(* CODESYS project tcunit.library
   Company: www.tcunit.org
   DefaultNamespace: TcUnit
   Version: 1.1.0.0
   Placeholder: TcUnit
   Author: Jakob Sagatowski and contributors
   Description: TwinCAT unit testing framework.
      Documentation and examples are available at www.tcunit.org
   Title: TcUnit

Project tree, tasks and I/O mapping:
  libraries: Base Interfaces, * (System); SysDir, * (System); SysFile, * (System); Tc2_Standard, * (Beckhoff Automation GmbH); Tc2_System, * (Beckhoff Automation GmbH); Tc2_Utilities, * (Beckhoff Automation GmbH)
  DUTs/
    data type E_AssertionType
    data type E_XmlError
    data type ST_AdsLogStringMessage
    data type ST_AssertArrayResult
    data type ST_AssertArrayResultInstances
    data type ST_AssertResult
    data type ST_AssertResultInstances
    data type ST_TestCaseResult
    data type ST_TestSuiteResult
    data type ST_TestSuiteResults
    data type U_ExpectedOrActual
  GVLs/
    global variables GVL_Param_TcUnit
    global variables GVL_TcUnit
  ITFs/
    interface I_AssertMessageFormatter: LogAssertFailure
    interface I_TestResultLogger: LogTestSuiteResults
    interface I_TestResults: GetAreTestResultsAvailable, GetTestSuiteResults
  POUs/
    Functions/
      WRITE_PROTECTED_/
        function WRITE_PROTECTED_BOOL [ST]
        function WRITE_PROTECTED_BYTE [ST]
        function WRITE_PROTECTED_DATE [ST]
        function WRITE_PROTECTED_DATE_AND_TIME [ST]
        function WRITE_PROTECTED_DINT [ST]
        function WRITE_PROTECTED_DWORD [ST]
        function WRITE_PROTECTED_INT [ST]
        function WRITE_PROTECTED_LINT [ST]
        function WRITE_PROTECTED_LREAL [ST]
        function WRITE_PROTECTED_LWORD [ST]
        function WRITE_PROTECTED_REAL [ST]
        function WRITE_PROTECTED_SINT [ST]
        function WRITE_PROTECTED_STRING [ST]
        function WRITE_PROTECTED_TIME [ST]
        function WRITE_PROTECTED_TIME_OF_DAY [ST]
        function WRITE_PROTECTED_UDINT [ST]
        function WRITE_PROTECTED_UINT [ST]
        function WRITE_PROTECTED_ULINT [ST]
        function WRITE_PROTECTED_USINT [ST]
        function WRITE_PROTECTED_WORD [ST]
        function WRITE_PROTECTED_WSTRING [ST]
      function F_AnyToUnionValue [ST]
      function F_AnyTypeClassToString [ST]
      function F_AssertionTypeToString [ST]
      function F_GetTestSuiteNameFromTestInstancePath [ST]
      function F_IsAnyEqualToUnionValue [ST]
      function F_RemoveInstancePathAndProjectNameFromTestInstancePath [ST]
      function IS_TEST_FINISHED [ST]
      function RUN [ST]
      function TEST [ST]
      function TEST_FINISHED [ST]
      function TEST_FINISHED_NAMED [ST]
    function block FB_AdjustAssertFailureMessageToMax253CharLength [ST]
    function block FB_AdsAssertMessageFormatter [ST]: LogAssertFailure
    function block FB_AdsLogStringMessageFifoQueue [ST]: GetAndRemoveLogFromQueue, GetLogCount, WriteLog
    function block FB_AdsTestResultLogger [ST]: FB_init, LogTestSuiteResults
    function block FB_AssertArrayResultStatic [ST]: AddAssertArrayResult, CopyDetectionCountAndResetDetectionCountInThisCycle, CreateAssertResultInstance, GetDetectionCount, GetDetectionCountThisCycle, GetNumberOfArrayAssertsForTest, ReportResult
    function block FB_AssertResultStatic [ST]: AddAssertResult, CopyDetectionCountAndResetDetectionCountInThisCycle, CreateAssertResultInstance, GetDetectionCount, GetDetectionCountThisCycle, GetNumberOfAssertsForTest, ReportResult
    function block FB_FileControl [ST]: Close, Delete, Open, Read, Write
    function block FB_StreamBuffer [ST]: Append, BufferSize, Clear, Copy, CutOff, Find, FindBack, Length, SetBuffer
    function block FB_TcUnitRunner [ST]: AbortRunningTestSuiteTests, RunTestSuiteTests
    function block FB_Test [ST]: GetAssertionMessage, GetAssertionType, GetName, GetNumberOfAssertions, IsFailed, IsFinished, IsSkipped, SetAssertionMessage, SetAssertionType, SetFailed, SetFinished, SetName, SetNumberOfAssertions, SetSkipped
    function block FB_TestResults [ST]: GetAreTestResultsAvailable, GetTestSuiteResults
    function block FB_TestSuite [ST]: AddTest, AddTestNameToInstancePath, AreAllTestsFinished, AssertArray2dEquals_LREAL, AssertArray2dEquals_REAL, AssertArray3dEquals_LREAL, AssertArray3dEquals_REAL, AssertArrayEquals_BOOL, AssertArrayEquals_BYTE, AssertArrayEquals_DINT, AssertArrayEquals_DWORD, AssertArrayEquals_INT, AssertArrayEquals_LINT, AssertArrayEquals_LREAL, AssertArrayEquals_LWORD, AssertArrayEquals_REAL, AssertArrayEquals_SINT, AssertArrayEquals_UDINT, AssertArrayEquals_UINT, AssertArrayEquals_ULINT, AssertArrayEquals_USINT, AssertArrayEquals_WORD, AssertEquals, AssertEquals_BOOL, AssertEquals_BYTE, AssertEquals_DATE, AssertEquals_DATE_AND_TIME, AssertEquals_DINT, AssertEquals_DWORD, AssertEquals_INT, AssertEquals_LINT, AssertEquals_LREAL, AssertEquals_LTIME, AssertEquals_LWORD, AssertEquals_REAL, AssertEquals_SINT, AssertEquals_STRING, AssertEquals_TIME, AssertEquals_TIME_OF_DAY, AssertEquals_UDINT, AssertEquals_UINT, AssertEquals_ULINT, AssertEquals_USINT, AssertEquals_WORD, AssertEquals_WSTRING, AssertFalse, AssertTrue, CalculateAndSetNumberOfAssertsForTest, FB_init, FindTestSuiteInstancePath, GetInstancePath, GetNumberOfFailedTests, GetNumberOfSkippedTests, GetNumberOfSuccessfulTests, GetNumberOfTests, GetTestByPosition, IsTestFinished, SetTestFailed, SetTestFinished
    function block FB_XmlControl [ST]: ClearBuffer, CloseTag, Length, NewComment, NewParameter, NewTag, NewTagData, SetBuffer, ToStartBuffer, WriteDocumentHeader
    function block FB_xUnitXmlPublisher [ST]: DeleteOpenWriteClose, FB_Init, Initialised, LogTestSuiteResults
  Version/
    global variables Global_Version
*)

// DUTs/E_AssertionType
{attribute 'qualified_only'}
{attribute 'strict'}
TYPE E_AssertionType :
(
    Type_UNDEFINED := 0,
    Type_ANY,

    (* Primitive types *)
    Type_BOOL,
    Type_BYTE,
    Type_DATE,
    Type_DATE_AND_TIME,
    Type_DINT,
    Type_DWORD,
    Type_INT,
    Type_LINT,
    Type_LREAL,
    Type_LTIME,
    Type_LWORD,
    Type_REAL,
    Type_SINT,
    Type_STRING,
    Type_TIME,
    Type_TIME_OF_DAY,
    Type_UDINT,
    Type_UINT,
    Type_ULINT,
    Type_USINT,
    Type_WORD,
    Type_WSTRING,

    (* Array types *)
    Type_Array2D_LREAL,
    Type_Array2D_REAL,
    Type_Array3D_LREAL,
    Type_Array3D_REAL,
    Type_Array_BOOL,
    Type_Array_BYTE,
    Type_Array_DINT,
    Type_Array_DWORD,
    Type_Array_INT,
    Type_Array_LINT,
    Type_Array_LREAL,
    Type_Array_LWORD,
    Type_Array_REAL,
    Type_Array_SINT,
    Type_Array_UDINT,
    Type_Array_UINT,
    Type_Array_ULINT,
    Type_Array_USINT,
    Type_Array_WORD
) BYTE;
END_TYPE

// DUTs/E_XmlError
{attribute 'qualified_only'}
{attribute 'strict'}
TYPE E_XmlError :
(
    Ok := 0,
    ErrorMaxBufferLen := 1,
    ErrorStringLen := 2,
    Error := 3
) BYTE;
END_TYPE

// DUTs/ST_AdsLogStringMessage
{attribute 'pack_mode' := '1'}
TYPE ST_AdsLogStringMessage :
STRUCT
	MsgCtrlMask : DWORD;
    MsgFmtStr : Tc2_System.T_MaxString;
    StrArg : Tc2_System.T_MaxString;
END_STRUCT
END_TYPE

// DUTs/ST_AssertArrayResult
TYPE ST_AssertArrayResult :
STRUCT
    ExpectedsSize : UDINT; // Size in bytes of the expecteds-array
    ExpectedsTypeClass : IBaseLibrary.TypeClass; // The data type of the expecteds-array
    ActualsSize : UDINT; // Size in bytes of the actuals-array
    ActualsTypeClass : IBaseLibrary.TypeClass; // The data type of the actuals-array
    Message : Tc2_System.T_MaxString;
    TestInstancePath : Tc2_System.T_MaxString;
END_STRUCT
END_TYPE

// DUTs/ST_AssertArrayResultInstances
TYPE ST_AssertArrayResultInstances :
STRUCT
    AssertArrayResult : ST_AssertArrayResult;
    DetectionCount : UINT; // Number of instances of the "AssertArrayResult"
    DetectionCountThisCycle : UINT; // Number of instance of the "AssertArrayResult" in this specific PLC-cycle
END_STRUCT
END_TYPE

// DUTs/ST_AssertResult
TYPE ST_AssertResult :
STRUCT
    Expected : U_ExpectedOrActual;
    Actual : U_ExpectedOrActual;
    Message : Tc2_System.T_MaxString;
    TestInstancePath : Tc2_System.T_MaxString;
END_STRUCT
END_TYPE

// DUTs/ST_AssertResultInstances
TYPE ST_AssertResultInstances :
STRUCT
    AssertResult : ST_AssertResult;
    DetectionCount : UINT; // Number of instances of the "AssertResult"
    DetectionCountThisCycle : UINT; // Number of instance of the "AssertResult" in this specific PLC-cycle
END_STRUCT
END_TYPE

// DUTs/ST_TestCaseResult
TYPE ST_TestCaseResult :
STRUCT
    TestName : Tc2_System.T_MaxString;
    TestClassName : Tc2_System.T_MaxString;
    TestIsFailed : BOOL;
    TestIsSkipped : BOOL;
    FailureMessage : Tc2_System.T_MaxString;
    FailureType : E_AssertionType;
    NumberOfAsserts : UINT;
END_STRUCT
END_TYPE

// DUTs/ST_TestSuiteResult
TYPE ST_TestSuiteResult :
STRUCT
    Name : Tc2_System.T_MaxString; // Full class name
    Identity : UINT(0..GVL_Param_TcUnit.MaxNumberOfTestSuites); // Should be 0..GVL_Param_TcUnit.MaxNumberOfTestSuites-1 but gives unknown compiler error
    NumberOfTests : UINT(0..GVL_Param_TcUnit.MaxNumberOfTestsForEachTestSuite);
    NumberOfFailedTests : UINT(0..GVL_Param_TcUnit.MaxNumberOfTestsForEachTestSuite);
    TestCaseResults : ARRAY[1..GVL_Param_TcUnit.MaxNumberOfTestsForEachTestSuite] OF ST_TestCaseResult;
END_STRUCT
END_TYPE

// DUTs/ST_TestSuiteResults
TYPE ST_TestSuiteResults :
STRUCT
    (* General test results *)
    NumberOfTestSuites : UINT; // The total number of test suites
    NumberOfTestCases : UINT; // The total number of test cases (for all test suites)
    NumberOfSuccessfulTestCases : UINT; // The total number of test cases that had all ASSERTS successful
    NumberOfFailedTestCases : UINT; // The total number of test cases that had at least one ASSERT failed

    (* Test results for each individiual test suite *)
    TestSuiteResults : ARRAY[1..GVL_Param_TcUnit.MaxNumberOfTestSuites] OF ST_TestSuiteResult;
END_STRUCT
END_TYPE

// DUTs/U_ExpectedOrActual
TYPE U_ExpectedOrActual :
UNION
    boolExpectedOrActual : BOOL;
    bitExpectedOrActual : BIT;
    byteExpectedOrActual : BYTE;
    dwordExpectedOrActual : DWORD;
    lwordExpectedOrActual : LWORD;
    stringExpectedOrActual : Tc2_System.T_MaxString;
    udintExpectedOrActual : UDINT;
    uintExpectedOrActual : UINT;
    usintExpectedOrActual : USINT;
    sintExpectedOrActual : SINT;
    intExpectedOrActual : INT;
    wordExpectedOrActual : WORD;
    dintExpectedOrActual : DINT;
    lintExpectedOrActual : LINT;
    ulintExpectedOrActual : ULINT;
    realExpectedOrActual : REAL;
    lrealExpectedOrActual : LREAL;
    wstringExpectedOrActual : WSTRING(255);
    timeExpectedOrActual : TIME;
    ltimeExpectedOrActual : LTIME;
    dateExpectedOrActual : DATE;
    dateandtimeExpectedOrActual : DATE_AND_TIME;
    timeofdayExpectedOrActual : TIME_OF_DAY;
END_UNION
END_TYPE

// GVLs/GVL_Param_TcUnit
{attribute 'qualified_only'}
VAR_GLOBAL CONSTANT
    MaxNumberOfTestSuites : UINT := 1000;
    MaxNumberOfTestsForEachTestSuite : UINT := 100;
    MaxNumberOfAssertsForEachTestSuite : UINT := 1000;

    (* TcUnit logs complete test results. These include:
         - Number of test suites
         - Number of tests
         - Number of successful tests
         - Number of failed tests
         - Any eventual failed assertion (with the expected & actual value plus an user defined message)
       These are all printed to the ADS logger (Visual Studio error list) marked with ERROR criticality

       On top of this TcUnit also reports some statistics/extended information with HINT/INFO criticality.
       These statistics are more detailed results of the tests. This information is used when results are
       being collected by an external software (such as TcUnit-Runner) to do for example Jenkins integration.
       This extra information however takes time to print, so by setting the following parameter to FALSE
       it will speed up TcUnit finishing. *)
    LogExtendedResults : BOOL := TRUE;

    (* Enable (TRUE) or disable (FALSE) publishing of the xUnit Xml report *)
    xUnitEnablePublish : BOOL := FALSE;

    (* Default reserved PLC memory buffer used for composition of the xUnit xml file (64 kb default) *)
    xUnitBufferSize : UDINT := 65535;

    (* Default path and filename for the xunit testresults e.g.: for use with jenkins *)
    xUnitFilePath : Tc2_System.T_MaxString := 'C:\tcunit_xunit_testresults.xml';

    (* This is the maximum number of ADS-messages that can be stored for reporting at the same time.
       Having a size of 2000 means that it's possible to report up to ~400 test cases in one single
       PLC cycle. Each entry consumes around 500 bytes, so with an example of a ring buffer size of
       2000 it means that TcUnit will consume around 1 MB of router memory. *) 
    AdsLogMessageFifoRingBufferSize : UINT := 2000;
END_VAR

// GVLs/GVL_TcUnit
{attribute 'no_assign'}
{attribute 'qualified_only'}
VAR_GLOBAL
    TcUnitRunner : FB_TcUnitRunner;

    (* Indication of whether the last instantiated test suite has an assert instance created *)
    TestSuiteIsRegistered : BOOL;

    (* Pointer to current test suite being called *)
    CurrentTestSuiteBeingCalled : POINTER TO FB_TestSuite;

    (* Current name of test being called *)
    CurrentTestNameBeingCalled : Tc2_System.T_MaxString;

    (* Whether or not the current test being called has finished running *)
    CurrentTestIsFinished : BOOL;

    (* This is a flag that indicates that the current test should be ignored, and
       thus that all assertions under it should be ignored as well. A test can be ignored either
       because the user has requested so, or because the test is a duplicate name *)
    IgnoreCurrentTest : BOOL;

    (* The assert function block instance should be 1:1 mapped to
       the test suite instance path. *)
    NumberOfInitializedTestSuites : UINT := 0;
    TestSuiteAddresses : ARRAY[1..GVL_Param_TcUnit.MaxNumberOfTestSuites] OF POINTER TO FB_TestSuite;

    (* Buffered ADS message queue for output to the error list *)
    AdsMessageQueue : FB_AdsLogStringMessageFifoQueue;
END_VAR

// Version/Global_Version
{attribute 'TcGenerated'}
{attribute 'no-analysis'}
{attribute 'linkalways'}
// This function has been automatically generated from the project information.
VAR_GLOBAL CONSTANT
	{attribute 'const_non_replaced'}
	stLibVersion_TcUnit : ST_LibVersion := (iMajor := 1, iMinor := 1, iBuild := 0, iRevision := 0, sVersion := '1.1.0.0');
END_VAR

// ITFs/I_AssertMessageFormatter
INTERFACE I_AssertMessageFormatter

METHOD LogAssertFailure
VAR_INPUT
    Expected : Tc2_System.T_MaxString;
    Actual : Tc2_System.T_MaxString;
    Message : Tc2_System.T_MaxString;
    TestInstancePath : Tc2_System.T_MaxString;
END_VAR
END_METHOD

END_INTERFACE

// ITFs/I_TestResultLogger
INTERFACE I_TestResultLogger

METHOD PUBLIC LogTestSuiteResults
END_METHOD

END_INTERFACE

// ITFs/I_TestResults
INTERFACE I_TestResults

METHOD GetAreTestResultsAvailable : BOOL
END_METHOD

METHOD GetTestSuiteResults : REFERENCE TO ST_TestSuiteResults;
END_METHOD

END_INTERFACE

// POUs/Functions/WRITE_PROTECTED_/WRITE_PROTECTED_BOOL
FUNCTION WRITE_PROTECTED_BOOL
VAR_INPUT
    Ptr : POINTER TO BOOL;
    Value : BOOL;
END_VAR

Ptr^ := Value;

END_FUNCTION

// POUs/Functions/WRITE_PROTECTED_/WRITE_PROTECTED_BYTE
FUNCTION WRITE_PROTECTED_BYTE
VAR_INPUT
    Ptr : POINTER TO BYTE;
    Value : BYTE;
END_VAR

Ptr^ := Value;

END_FUNCTION

// POUs/Functions/WRITE_PROTECTED_/WRITE_PROTECTED_DATE
FUNCTION WRITE_PROTECTED_DATE
VAR_INPUT
    Ptr : POINTER TO DATE;
    Value : DATE;
END_VAR

Ptr^ := Value;

END_FUNCTION

// POUs/Functions/WRITE_PROTECTED_/WRITE_PROTECTED_DATE_AND_TIME
FUNCTION WRITE_PROTECTED_DATE_AND_TIME
VAR_INPUT
    Ptr : POINTER TO DATE_AND_TIME;
    Value : DATE_AND_TIME;
END_VAR

Ptr^ := Value;

END_FUNCTION

// POUs/Functions/WRITE_PROTECTED_/WRITE_PROTECTED_DINT
FUNCTION WRITE_PROTECTED_DINT
VAR_INPUT
    Ptr : POINTER TO DINT;
    Value : DINT;
END_VAR

Ptr^ := Value;

END_FUNCTION

// POUs/Functions/WRITE_PROTECTED_/WRITE_PROTECTED_DWORD
FUNCTION WRITE_PROTECTED_DWORD
VAR_INPUT
    Ptr : POINTER TO DWORD;
    Value : DWORD;
END_VAR

Ptr^ := Value;

END_FUNCTION

// POUs/Functions/WRITE_PROTECTED_/WRITE_PROTECTED_INT
FUNCTION WRITE_PROTECTED_INT
VAR_INPUT
    Ptr : POINTER TO INT;
    Value : INT;
END_VAR

Ptr^ := Value;

END_FUNCTION

// POUs/Functions/WRITE_PROTECTED_/WRITE_PROTECTED_LINT
FUNCTION WRITE_PROTECTED_LINT
VAR_INPUT
    Ptr : POINTER TO LINT;
    Value : LINT;
END_VAR

Ptr^ := Value;

END_FUNCTION

// POUs/Functions/WRITE_PROTECTED_/WRITE_PROTECTED_LREAL
FUNCTION WRITE_PROTECTED_LREAL
VAR_INPUT
    Ptr : POINTER TO LREAL;
    Value : LREAL;
END_VAR

Ptr^ := Value;

END_FUNCTION

// POUs/Functions/WRITE_PROTECTED_/WRITE_PROTECTED_LWORD
FUNCTION WRITE_PROTECTED_LWORD
VAR_INPUT
    Ptr : POINTER TO LWORD;
    Value : LWORD;
END_VAR

Ptr^ := Value;

END_FUNCTION

// POUs/Functions/WRITE_PROTECTED_/WRITE_PROTECTED_REAL
FUNCTION WRITE_PROTECTED_REAL
VAR_INPUT
    Ptr : POINTER TO REAL;
    Value : REAL;
END_VAR

Ptr^ := Value;

END_FUNCTION

// POUs/Functions/WRITE_PROTECTED_/WRITE_PROTECTED_SINT
FUNCTION WRITE_PROTECTED_SINT
VAR_INPUT
    Ptr : POINTER TO SINT;
    Value : SINT;
END_VAR

Ptr^ := Value;

END_FUNCTION

// POUs/Functions/WRITE_PROTECTED_/WRITE_PROTECTED_STRING
FUNCTION WRITE_PROTECTED_STRING
VAR_INPUT
    Ptr : POINTER TO STRING;
    Value : STRING;
END_VAR

Ptr^ := Value;

END_FUNCTION

// POUs/Functions/WRITE_PROTECTED_/WRITE_PROTECTED_TIME
FUNCTION WRITE_PROTECTED_TIME
VAR_INPUT
    Ptr : POINTER TO TIME;
    Value : TIME;
END_VAR

Ptr^ := Value;

END_FUNCTION

// POUs/Functions/WRITE_PROTECTED_/WRITE_PROTECTED_TIME_OF_DAY
FUNCTION WRITE_PROTECTED_TIME_OF_DAY
VAR_INPUT
    Ptr : POINTER TO TIME_OF_DAY;
    Value : TIME_OF_DAY;
END_VAR

Ptr^ := Value;

END_FUNCTION

// POUs/Functions/WRITE_PROTECTED_/WRITE_PROTECTED_UDINT
FUNCTION WRITE_PROTECTED_UDINT
VAR_INPUT
    Ptr : POINTER TO UDINT;
    Value : UDINT;
END_VAR

Ptr^ := Value;

END_FUNCTION

// POUs/Functions/WRITE_PROTECTED_/WRITE_PROTECTED_UINT
FUNCTION WRITE_PROTECTED_UINT
VAR_INPUT
    Ptr : POINTER TO UINT;
    Value : UINT;
END_VAR

Ptr^ := Value;

END_FUNCTION

// POUs/Functions/WRITE_PROTECTED_/WRITE_PROTECTED_ULINT
FUNCTION WRITE_PROTECTED_ULINT
VAR_INPUT
    Ptr : POINTER TO ULINT;
    Value : ULINT;
END_VAR

Ptr^ := Value;

END_FUNCTION

// POUs/Functions/WRITE_PROTECTED_/WRITE_PROTECTED_USINT
FUNCTION WRITE_PROTECTED_USINT
VAR_INPUT
    Ptr : POINTER TO USINT;
    Value : USINT;
END_VAR

Ptr^ := Value;

END_FUNCTION

// POUs/Functions/WRITE_PROTECTED_/WRITE_PROTECTED_WORD
FUNCTION WRITE_PROTECTED_WORD
VAR_INPUT
    Ptr : POINTER TO WORD;
    Value : WORD;
END_VAR

Ptr^ := Value;

END_FUNCTION

// POUs/Functions/WRITE_PROTECTED_/WRITE_PROTECTED_WSTRING
FUNCTION WRITE_PROTECTED_WSTRING
VAR_INPUT
    Ptr : POINTER TO WSTRING;
    Value : WSTRING;
END_VAR

Ptr^ := Value;

END_FUNCTION

// POUs/Functions/F_AnyToUnionValue
FUNCTION F_AnyToUnionValue : U_ExpectedOrActual
VAR_INPUT
    AnySize : UDINT;
    AnyTypeClass : IBaseLibrary.TypeClass;
    AnyValue : POINTER TO BYTE;
END_VAR

CASE AnyTypeClass OF
    IBaseLibrary.TypeClass.TYPE_BOOL :
        Tc2_System.MEMCPY(destaddr := ADR(F_AnyToUnionValue.boolExpectedOrActual),
                          srcAddr := AnyValue,
                          n := AnySize);

    IBaseLibrary.TypeClass.TYPE_BIT :
        {warning disable C0355}
        Tc2_System.MEMCPY(destaddr := ADR(F_AnyToUnionValue.bitExpectedOrActual),
                          srcAddr := AnyValue,
                          n := AnySize);
        {warning enable C0355}

    IBaseLibrary.TypeClass.TYPE_BYTE :
        Tc2_System.MEMCPY(destaddr := ADR(F_AnyToUnionValue.byteExpectedOrActual),
                          srcAddr := AnyValue,
                          n := AnySize);

    IBaseLibrary.TypeClass.TYPE_WORD :
        Tc2_System.MEMCPY(destaddr := ADR(F_AnyToUnionValue.wordExpectedOrActual),
                          srcAddr := AnyValue,
                          n := AnySize);

    IBaseLibrary.TypeClass.TYPE_DWORD :
        Tc2_System.MEMCPY(destaddr := ADR(F_AnyToUnionValue.dwordExpectedOrActual),
                          srcAddr := AnyValue,
                          n := AnySize);

    IBaseLibrary.TypeClass.TYPE_LWORD :
        Tc2_System.MEMCPY(destaddr := ADR(F_AnyToUnionValue.lwordExpectedOrActual),
                          srcAddr := AnyValue,
                          n := AnySize);

    IBaseLibrary.TypeClass.TYPE_SINT :
        Tc2_System.MEMCPY(destaddr := ADR(F_AnyToUnionValue.sintExpectedOrActual),
                          srcAddr := AnyValue,
                          n := AnySize);

    IBaseLibrary.TypeClass.TYPE_INT :
        Tc2_System.MEMCPY(destaddr := ADR(F_AnyToUnionValue.intExpectedOrActual),
                          srcAddr := AnyValue,
                          n := AnySize);

    IBaseLibrary.TypeClass.TYPE_DINT :
        Tc2_System.MEMCPY(destaddr := ADR(F_AnyToUnionValue.dintExpectedOrActual),
                          srcAddr := AnyValue,
                          n := AnySize);

    IBaseLibrary.TypeClass.TYPE_LINT :
        Tc2_System.MEMCPY(destaddr := ADR(F_AnyToUnionValue.lintExpectedOrActual),
                          srcAddr := AnyValue,
                          n := AnySize);

    IBaseLibrary.TypeClass.TYPE_USINT :
        Tc2_System.MEMCPY(destaddr := ADR(F_AnyToUnionValue.usintExpectedOrActual),
                          srcAddr := AnyValue,
                          n := AnySize);

    IBaseLibrary.TypeClass.TYPE_UINT :
        Tc2_System.MEMCPY(destaddr := ADR(F_AnyToUnionValue.uintExpectedOrActual),
                          srcAddr := AnyValue,
                          n := AnySize);

    IBaseLibrary.TypeClass.TYPE_UDINT :
        Tc2_System.MEMCPY(destaddr := ADR(F_AnyToUnionValue.udintExpectedOrActual),
                          srcAddr := AnyValue,
                          n := AnySize);

    IBaseLibrary.TypeClass.TYPE_ULINT :
        Tc2_System.MEMCPY(destaddr := ADR(F_AnyToUnionValue.ulintExpectedOrActual),
                          srcAddr := AnyValue,
                          n := AnySize);

    IBaseLibrary.TypeClass.TYPE_REAL :
        Tc2_System.MEMCPY(destaddr := ADR(F_AnyToUnionValue.realExpectedOrActual),
                          srcAddr := AnyValue,
                          n := AnySize);

    IBaseLibrary.TypeClass.TYPE_LREAL :
        Tc2_System.MEMCPY(destaddr := ADR(F_AnyToUnionValue.lrealExpectedOrActual),
                          srcAddr := AnyValue,
                          n := AnySize);

    IBaseLibrary.TypeClass.TYPE_STRING :
        Tc2_System.MEMCPY(destaddr := ADR(F_AnyToUnionValue.stringExpectedOrActual),
                          srcAddr := AnyValue,
                          n := AnySize);

    IBaseLibrary.TypeClass.TYPE_WSTRING :
        Tc2_System.MEMCPY(destaddr := ADR(F_AnyToUnionValue.wstringExpectedOrActual),
                          srcAddr := AnyValue,
                          n := AnySize);

    IBaseLibrary.TypeClass.TYPE_TIME :
        Tc2_System.MEMCPY(destaddr := ADR(F_AnyToUnionValue.timeExpectedOrActual),
                          srcAddr := AnyValue,
                          n := AnySize);

    IBaseLibrary.TypeClass.TYPE_DATE :
        Tc2_System.MEMCPY(destaddr := ADR(F_AnyToUnionValue.dateExpectedOrActual),
                          srcAddr := AnyValue,
                          n := AnySize);

    IBaseLibrary.TypeClass.TYPE_DATEANDTIME :
        Tc2_System.MEMCPY(destaddr := ADR(F_AnyToUnionValue.dateandtimeExpectedOrActual),
                          srcAddr := AnyValue,
                          n := AnySize);

    IBaseLibrary.TypeClass.TYPE_TIMEOFDAY :
        Tc2_System.MEMCPY(destaddr := ADR(F_AnyToUnionValue.timeofdayExpectedOrActual),
                          srcAddr := AnyValue,
                          n := AnySize);

    IBaseLibrary.TypeClass.TYPE_POINTER :
        (* None *)

    IBaseLibrary.TypeClass.TYPE_REFERENCE :
        (* None *)

    IBaseLibrary.TypeClass.TYPE_SUBRANGE :
        (* None *)

    IBaseLibrary.TypeClass.TYPE_ENUM :
        (* None *)

    IBaseLibrary.TypeClass.TYPE_ARRAY :
        (* None *)

    IBaseLibrary.TypeClass.TYPE_PARAMS :
        (* None *)

    IBaseLibrary.TypeClass.TYPE_USERDEF :
        (* None *)

    IBaseLibrary.TypeClass.TYPE_NONE :
        (* None *)

    IBaseLibrary.TypeClass.TYPE_ANY :
        (* None *)

    IBaseLibrary.TypeClass.TYPE_ANYBIT :
        (* None *)

    IBaseLibrary.TypeClass.TYPE_ANYDATE :
        (* None *)

    IBaseLibrary.TypeClass.TYPE_ANYINT :
        (* None *)

    IBaseLibrary.TypeClass.TYPE_ANYNUM :
        (* None *)

    IBaseLibrary.TypeClass.TYPE_ANYREAL :
        (* None *)

    IBaseLibrary.TypeClass.TYPE_LAZY :
        (* None *)

    IBaseLibrary.TypeClass.TYPE_LTIME :
        Tc2_System.MEMCPY(destaddr := ADR(F_AnyToUnionValue.ltimeExpectedOrActual),
                          srcAddr := AnyValue,
                          n := AnySize);

    IBaseLibrary.TypeClass.TYPE_BITCONST :
        (* None *)

    IBaseLibrary.TypeClass.TYPE_INTERFACE :
        (* None *)

    ELSE
        (* None *)
END_CASE

END_FUNCTION

// POUs/Functions/F_AnyTypeClassToString
(*
    This function takes the type-class of a ANY-variable and returns the STRING representation of it.
*)
FUNCTION F_AnyTypeClassToString : STRING
VAR_INPUT
    AnyTypeClass : __SYSTEM.TYPE_CLASS;
END_VAR

CASE UDINT_TO_INT(AnyTypeClass) OF
    IBaseLibrary.TypeClass.TYPE_BOOL :
        F_AnyTypeClassToString := 'BOOL';
    IBaseLibrary.TypeClass.TYPE_BIT :
        F_AnyTypeClassToString := 'BIT';
    IBaseLibrary.TypeClass.TYPE_BYTE :
        F_AnyTypeClassToString := 'BYTE';
    IBaseLibrary.TypeClass.TYPE_WORD :
        F_AnyTypeClassToString := 'WORD';
    IBaseLibrary.TypeClass.TYPE_DWORD :
        F_AnyTypeClassToString := 'DWORD';
    IBaseLibrary.TypeClass.TYPE_LWORD :
        F_AnyTypeClassToString := 'LWORD';
    IBaseLibrary.TypeClass.TYPE_SINT :
        F_AnyTypeClassToString := 'SINT';
    IBaseLibrary.TypeClass.TYPE_INT :
        F_AnyTypeClassToString := 'INT';
    IBaseLibrary.TypeClass.TYPE_DINT :
        F_AnyTypeClassToString := 'DINT';
    IBaseLibrary.TypeClass.TYPE_LINT :
        F_AnyTypeClassToString := 'LINT';
    IBaseLibrary.TypeClass.TYPE_USINT :
        F_AnyTypeClassToString := 'USINT';
    IBaseLibrary.TypeClass.TYPE_UINT :
        F_AnyTypeClassToString := 'UINT';
    IBaseLibrary.TypeClass.TYPE_UDINT :
        F_AnyTypeClassToString := 'UDINT';
    IBaseLibrary.TypeClass.TYPE_ULINT :
        F_AnyTypeClassToString := 'ULINT';
    IBaseLibrary.TypeClass.TYPE_REAL :
        F_AnyTypeClassToString := 'REAL';
    IBaseLibrary.TypeClass.TYPE_LREAL :
        F_AnyTypeClassToString := 'LREAL';
    IBaseLibrary.TypeClass.TYPE_STRING :
        F_AnyTypeClassToString := 'STRING';
    IBaseLibrary.TypeClass.TYPE_WSTRING :
        F_AnyTypeClassToString := 'WSTRING';
    IBaseLibrary.TypeClass.TYPE_TIME :
        F_AnyTypeClassToString := 'TIME';
    IBaseLibrary.TypeClass.TYPE_DATE :
        F_AnyTypeClassToString := 'DATE';
    IBaseLibrary.TypeClass.TYPE_DATEANDTIME :
        F_AnyTypeClassToString := 'DATEANDTIME';
    IBaseLibrary.TypeClass.TYPE_TIMEOFDAY :
        F_AnyTypeClassToString := 'TIMEOFDAY';
    IBaseLibrary.TypeClass.TYPE_POINTER :
        F_AnyTypeClassToString := 'POINTER';
    IBaseLibrary.TypeClass.TYPE_REFERENCE :
        F_AnyTypeClassToString := 'REFERENCE';
    IBaseLibrary.TypeClass.TYPE_SUBRANGE :
        F_AnyTypeClassToString := 'SUBRANGE';
    IBaseLibrary.TypeClass.TYPE_ENUM :
        F_AnyTypeClassToString := 'ENUM';
    IBaseLibrary.TypeClass.TYPE_ARRAY :
        F_AnyTypeClassToString := 'ARRAY';
    IBaseLibrary.TypeClass.TYPE_PARAMS :
        F_AnyTypeClassToString := 'PARAMS';
    IBaseLibrary.TypeClass.TYPE_USERDEF :
        F_AnyTypeClassToString := 'USERDEF';
    IBaseLibrary.TypeClass.TYPE_NONE :
        F_AnyTypeClassToString := 'NONE';
    IBaseLibrary.TypeClass.TYPE_ANY :
        F_AnyTypeClassToString := 'ANY';
    IBaseLibrary.TypeClass.TYPE_ANYBIT :
        F_AnyTypeClassToString := 'ANYBIT';
    IBaseLibrary.TypeClass.TYPE_ANYDATE :
        F_AnyTypeClassToString := 'ANYDATE';
    IBaseLibrary.TypeClass.TYPE_ANYINT :
        F_AnyTypeClassToString := 'ANYINT';
    IBaseLibrary.TypeClass.TYPE_ANYNUM :
        F_AnyTypeClassToString := 'ANYNUM';
    IBaseLibrary.TypeClass.TYPE_ANYREAL :
        F_AnyTypeClassToString := 'ANYREAL';
    IBaseLibrary.TypeClass.TYPE_LAZY :
        F_AnyTypeClassToString := 'LAZY';
    IBaseLibrary.TypeClass.TYPE_LTIME :
        F_AnyTypeClassToString := 'LTIME';
    IBaseLibrary.TypeClass.TYPE_BITCONST :
        F_AnyTypeClassToString := 'BITCONST';
    IBaseLibrary.TypeClass.TYPE_INTERFACE :
        F_AnyTypeClassToString := 'INTERFACE';
    ELSE
        F_AnyTypeClassToString := 'UNKNOWN';
END_CASE

END_FUNCTION

// POUs/Functions/F_AssertionTypeToString
(* Since TwinCAT 3.1.4024.x it's possible to do TO_STRING on enumerations,
   but for backward compability we need to do it manually *)
FUNCTION F_AssertionTypeToString : Tc2_System.T_MaxString
VAR_INPUT
    AssertionType : E_AssertionType;
END_VAR

CASE AssertionType OF
    E_AssertionType.Type_UNDEFINED :
        F_AssertionTypeToString := 'UNDEFINED';
    E_AssertionType.Type_ANY :
        F_AssertionTypeToString := 'ANY';

    (* Primitive types *)
    E_AssertionType.Type_BOOL :
        F_AssertionTypeToString := 'BOOL';
    E_AssertionType.Type_BYTE :
        F_AssertionTypeToString := 'BYTE';
    E_AssertionType.Type_DATE :
        F_AssertionTypeToString := 'DATE';
    E_AssertionType.Type_DATE_AND_TIME :
        F_AssertionTypeToString := 'DATE_AND_TIME';
    E_AssertionType.Type_DINT :
        F_AssertionTypeToString := 'DINT';
    E_AssertionType.Type_DWORD :
        F_AssertionTypeToString := 'DWORD';
    E_AssertionType.Type_INT :
        F_AssertionTypeToString := 'INT';
    E_AssertionType.Type_LINT :
        F_AssertionTypeToString := 'LINT';
    E_AssertionType.Type_LREAL :
        F_AssertionTypeToString := 'LREAL';
    E_AssertionType.Type_LTIME :
        F_AssertionTypeToString := 'LTIME';
    E_AssertionType.Type_LWORD :
        F_AssertionTypeToString := 'LWORD';
    E_AssertionType.Type_REAL :
        F_AssertionTypeToString := 'REAL';
    E_AssertionType.Type_SINT :
        F_AssertionTypeToString := 'SINT';
    E_AssertionType.Type_STRING :
        F_AssertionTypeToString := 'STRING';
    E_AssertionType.Type_TIME :
        F_AssertionTypeToString := 'TIME';
    E_AssertionType.Type_TIME_OF_DAY :
        F_AssertionTypeToString := 'TIME_OF_DAY';
    E_AssertionType.Type_UDINT :
        F_AssertionTypeToString := 'UDINT';
    E_AssertionType.Type_UINT :
        F_AssertionTypeToString := 'UINT';
    E_AssertionType.Type_ULINT :
        F_AssertionTypeToString := 'ULINT';
    E_AssertionType.Type_USINT :
        F_AssertionTypeToString := 'USINT';
    E_AssertionType.Type_WORD :
        F_AssertionTypeToString := 'WORD';
    E_AssertionType.Type_WSTRING :
        F_AssertionTypeToString := 'WSTRING';


    (* Array types *)
    E_AssertionType.Type_Array2D_LREAL :
        F_AssertionTypeToString := 'Array2D_LREAL';
    E_AssertionType.Type_Array2D_REAL :
        F_AssertionTypeToString := 'Array2D_REAL';
    E_AssertionType.Type_Array3D_LREAL :
        F_AssertionTypeToString := 'Array3D_LREAL';
    E_AssertionType.Type_Array3D_REAL :
        F_AssertionTypeToString := 'Array3D_REAL';
    E_AssertionType.Type_Array_BOOL :
        F_AssertionTypeToString := 'Array_BOOL';
    E_AssertionType.Type_Array_BYTE :
        F_AssertionTypeToString := 'Array_BYTE';
    E_AssertionType.Type_Array_DINT :
        F_AssertionTypeToString := 'Array_DINT';
    E_AssertionType.Type_Array_DWORD :
        F_AssertionTypeToString := 'Array_DWORD';
    E_AssertionType.Type_Array_INT :
        F_AssertionTypeToString := 'Array_INT';
    E_AssertionType.Type_Array_LINT :
        F_AssertionTypeToString := 'Array_LINT';
    E_AssertionType.Type_Array_LREAL :
        F_AssertionTypeToString := 'Array_LREAL';
    E_AssertionType.Type_Array_LWORD :
        F_AssertionTypeToString := 'Array_LWORD';
    E_AssertionType.Type_Array_REAL :
        F_AssertionTypeToString := 'Array_REAL';
    E_AssertionType.Type_Array_SINT :
        F_AssertionTypeToString := 'Array_SINT';
    E_AssertionType.Type_Array_UDINT :
        F_AssertionTypeToString := 'Array_UDINT';
    E_AssertionType.Type_Array_UINT :
        F_AssertionTypeToString := 'Array_UINT';
    E_AssertionType.Type_Array_ULINT :
        F_AssertionTypeToString := 'Array_ULINT';
    E_AssertionType.Type_Array_USINT :
        F_AssertionTypeToString := 'Array_USINT';
    E_AssertionType.Type_Array_WORD :
        F_AssertionTypeToString := 'Array_WORD';

    ELSE
        F_AssertionTypeToString := 'UNDEFINED';

END_CASE

END_FUNCTION

// POUs/Functions/F_GetTestSuiteNameFromTestInstancePath
FUNCTION F_GetTestSuiteNameFromTestInstancePath : Tc2_System.T_MaxString
VAR_INPUT
    TestInstancePath : Tc2_System.T_MaxString;
END_VAR
VAR
    TestSuiteName : Tc2_System.T_MaxString;
    FindPosition : INT;
END_VAR

TestSuiteName := F_RemoveInstancePathAndProjectNameFromTestInstancePath(TestInstancePath := TestInstancePath);
(* Remove everything except the test suite name *)
FindPosition := Tc2_Standard.FIND(STR1 := TestSuiteName, '.');
TestSuiteName := Tc2_Standard.RIGHT(STR := TestSuiteName, SIZE := Tc2_Standard.LEN(STR := TestSuiteName) - FindPosition);
F_GetTestSuiteNameFromTestInstancePath := TestSuiteName;

END_FUNCTION

// POUs/Functions/F_RemoveInstancePathAndProjectNameFromTestInstancePath
FUNCTION F_RemoveInstancePathAndProjectNameFromTestInstancePath : Tc2_System.T_MaxString
VAR_INPUT
    TestInstancePath : Tc2_System.T_MaxString;
END_VAR
VAR
    CharacterPositionOfProjectName : INT;
    ProjectNameWithDot : Tc2_System.T_MaxString;
END_VAR

(* Add the '.' character to the project name for search *)
ProjectNameWithDot := Tc2_Standard.CONCAT(STR1 := TwinCAT_SystemInfoVarList._AppInfo.ProjectName, STR2 := '.');

(* Find the character position of the beginning of the first occurence of the project name *)
CharacterPositionOfProjectName := Tc2_Standard.FIND(STR1 := TestInstancePath, STR2 := ProjectNameWithDot);

IF CharacterPositionOfProjectName > 0 THEN
    TestInstancePath := Tc2_Standard.DELETE(STR := TestInstancePath,
                                            LEN := CharacterPositionOfProjectName-1 + Tc2_Standard.LEN(ProjectNameWithDot),
                                            POS := 1);
END_IF

(* Check if the project name happens to be the same as namespace, and in that case, remove that as well *)
CharacterPositionOfProjectName := Tc2_Standard.FIND(STR1 := TestInstancePath,
                                                    STR2 := ProjectNameWithDot);

IF CharacterPositionOfProjectName > 0 THEN
    TestInstancePath := Tc2_Standard.DELETE(STR := TestInstancePath,
                                            LEN := CharacterPositionOfProjectName - 1 + 
                                                Tc2_Standard.LEN(STR := ProjectNameWithDot),
                                            POS := 1);
END_IF

F_RemoveInstancePathAndProjectNameFromTestInstancePath := TestInstancePath;

END_FUNCTION

// POUs/Functions/TEST
(*
    This function declares a new test (if it has not been already declared in an earlier cycle)
*)
FUNCTION TEST
VAR_INPUT
    TestName : Tc2_System.T_MaxString;
END_VAR
VAR
    CounterTestSuiteAddress : UINT;
END_VAR

(* Mark this test as the current one being executed *)
GVL_TcUnit.CurrentTestNameBeingCalled := TestName;

(* Check if combination of address for the test suite and test name already exists.
   For every test suite the name of the test case needs to be unique.
   If a test with this name already exists, don't add it to the available tests.
   Otherwise, add it to the available tests *)

FOR CounterTestSuiteAddress := 1 TO GVL_TcUnit.NumberOfInitializedTestSuites BY 1 DO
    (* Look for the test suite by comparing to the one that is currently running *)
    IF GVL_TcUnit.TestSuiteAddresses[CounterTestSuiteAddress] = GVL_TcUnit.CurrentTestSuiteBeingCalled THEN
        GVL_TcUnit.TestSuiteAddresses[CounterTestSuiteAddress]^.AddTest(TestName := TestName);
        GVL_TcUnit.CurrentTestIsFinished := GVL_TcUnit.TestSuiteAddresses[CounterTestSuiteAddress]^.IsTestFinished(TestName := TestName);
        RETURN;
    END_IF
END_FOR

END_FUNCTION

// POUs/Functions/F_IsAnyEqualToUnionValue
FUNCTION F_IsAnyEqualToUnionValue : BOOL
VAR_INPUT
    uExpectedOrActual : U_ExpectedOrActual;
    ExpectedOrActualSize : UDINT;
    ExpectedOrActualTypeClass : IBaseLibrary.TypeClass;
    ExpectedOrActualValue : POINTER TO BYTE;
END_VAR
VAR
    AnyExpectedOrActual : U_ExpectedOrActual;
END_VAR

AnyExpectedOrActual := F_AnyToUnionValue(AnySize := ExpectedOrActualSize,
                                         AnyTypeClass := ExpectedOrActualTypeClass,
                                         AnyValue := ExpectedOrActualValue);

CASE ExpectedOrActualTypeClass OF

    IBaseLibrary.TypeClass.TYPE_BOOL :
        F_IsAnyEqualToUnionValue := uExpectedOrActual.boolExpectedOrActual = AnyExpectedOrActual.boolExpectedOrActual;

    IBaseLibrary.TypeClass.TYPE_BIT :
        F_IsAnyEqualToUnionValue := uExpectedOrActual.bitExpectedOrActual = AnyExpectedOrActual.bitExpectedOrActual;

    IBaseLibrary.TypeClass.TYPE_BYTE :
        F_IsAnyEqualToUnionValue := uExpectedOrActual.byteExpectedOrActual = AnyExpectedOrActual.byteExpectedOrActual;

    IBaseLibrary.TypeClass.TYPE_WORD :
        F_IsAnyEqualToUnionValue := uExpectedOrActual.wordExpectedOrActual = AnyExpectedOrActual.wordExpectedOrActual;

    IBaseLibrary.TypeClass.TYPE_DWORD :
        F_IsAnyEqualToUnionValue := uExpectedOrActual.dwordExpectedOrActual = AnyExpectedOrActual.dwordExpectedOrActual;

    IBaseLibrary.TypeClass.TYPE_LWORD :
        F_IsAnyEqualToUnionValue := uExpectedOrActual.lwordExpectedOrActual = AnyExpectedOrActual.lwordExpectedOrActual;

    IBaseLibrary.TypeClass.TYPE_SINT :
        F_IsAnyEqualToUnionValue := uExpectedOrActual.sintExpectedOrActual = AnyExpectedOrActual.sintExpectedOrActual;

    IBaseLibrary.TypeClass.TYPE_INT :
        F_IsAnyEqualToUnionValue := uExpectedOrActual.intExpectedOrActual = AnyExpectedOrActual.intExpectedOrActual;

    IBaseLibrary.TypeClass.TYPE_DINT :
        F_IsAnyEqualToUnionValue := uExpectedOrActual.dintExpectedOrActual = AnyExpectedOrActual.dintExpectedOrActual;

    IBaseLibrary.TypeClass.TYPE_LINT :
        F_IsAnyEqualToUnionValue := uExpectedOrActual.lintExpectedOrActual = AnyExpectedOrActual.lintExpectedOrActual;

    IBaseLibrary.TypeClass.TYPE_USINT :
        F_IsAnyEqualToUnionValue := uExpectedOrActual.usintExpectedOrActual = AnyExpectedOrActual.usintExpectedOrActual;

    IBaseLibrary.TypeClass.TYPE_UINT :
        F_IsAnyEqualToUnionValue := uExpectedOrActual.uintExpectedOrActual = AnyExpectedOrActual.uintExpectedOrActual;

    IBaseLibrary.TypeClass.TYPE_UDINT :
        F_IsAnyEqualToUnionValue := uExpectedOrActual.udintExpectedOrActual = AnyExpectedOrActual.udintExpectedOrActual;

    IBaseLibrary.TypeClass.TYPE_ULINT :
        F_IsAnyEqualToUnionValue := uExpectedOrActual.ulintExpectedOrActual = AnyExpectedOrActual.ulintExpectedOrActual;

    IBaseLibrary.TypeClass.TYPE_REAL :
        F_IsAnyEqualToUnionValue := uExpectedOrActual.realExpectedOrActual = AnyExpectedOrActual.realExpectedOrActual;

    IBaseLibrary.TypeClass.TYPE_LREAL :
        F_IsAnyEqualToUnionValue := uExpectedOrActual.lrealExpectedOrActual = AnyExpectedOrActual.lrealExpectedOrActual;

    IBaseLibrary.TypeClass.TYPE_STRING :
        F_IsAnyEqualToUnionValue := uExpectedOrActual.stringExpectedOrActual = AnyExpectedOrActual.stringExpectedOrActual;

    IBaseLibrary.TypeClass.TYPE_WSTRING :
        F_IsAnyEqualToUnionValue := uExpectedOrActual.wstringExpectedOrActual = AnyExpectedOrActual.wstringExpectedOrActual;

    IBaseLibrary.TypeClass.TYPE_TIME :
        F_IsAnyEqualToUnionValue := uExpectedOrActual.timeExpectedOrActual = AnyExpectedOrActual.timeExpectedOrActual;

    IBaseLibrary.TypeClass.TYPE_DATE :
        F_IsAnyEqualToUnionValue := uExpectedOrActual.dateExpectedOrActual = AnyExpectedOrActual.dateExpectedOrActual;

    IBaseLibrary.TypeClass.TYPE_DATEANDTIME :
        F_IsAnyEqualToUnionValue := uExpectedOrActual.dateandtimeExpectedOrActual = AnyExpectedOrActual.dateandtimeExpectedOrActual;

    IBaseLibrary.TypeClass.TYPE_TIMEOFDAY :
        F_IsAnyEqualToUnionValue := uExpectedOrActual.timeofdayExpectedOrActual = AnyExpectedOrActual.timeofdayExpectedOrActual;

    IBaseLibrary.TypeClass.TYPE_POINTER :
        F_IsAnyEqualToUnionValue := FALSE;

    IBaseLibrary.TypeClass.TYPE_REFERENCE :
        F_IsAnyEqualToUnionValue := FALSE;

    IBaseLibrary.TypeClass.TYPE_SUBRANGE :
        F_IsAnyEqualToUnionValue := FALSE;

    IBaseLibrary.TypeClass.TYPE_ENUM :
        F_IsAnyEqualToUnionValue := FALSE;

    IBaseLibrary.TypeClass.TYPE_ARRAY :
        F_IsAnyEqualToUnionValue := FALSE;

    IBaseLibrary.TypeClass.TYPE_PARAMS :
        F_IsAnyEqualToUnionValue := FALSE;

    IBaseLibrary.TypeClass.TYPE_USERDEF :
        F_IsAnyEqualToUnionValue := FALSE;

    IBaseLibrary.TypeClass.TYPE_NONE :
        F_IsAnyEqualToUnionValue := FALSE;

    IBaseLibrary.TypeClass.TYPE_ANY :
        (* Even though the data input of the ExpectedOrActual is ANY, this CASE-switch will never
           enter this case, but instead the type-class that it is an instance of. So for instance,
           if the ExpectedOrActual is an instance of INT, this case-switch will enter the 
           IBaseLibrary.TypeClass.TYPE_INT case. *)
        F_IsAnyEqualToUnionValue := FALSE;

    IBaseLibrary.TypeClass.TYPE_ANYBIT :
        F_IsAnyEqualToUnionValue := FALSE;

    IBaseLibrary.TypeClass.TYPE_ANYDATE :
        F_IsAnyEqualToUnionValue := FALSE;

    IBaseLibrary.TypeClass.TYPE_ANYINT :
        F_IsAnyEqualToUnionValue := FALSE;

    IBaseLibrary.TypeClass.TYPE_ANYNUM :
        F_IsAnyEqualToUnionValue := FALSE;

    IBaseLibrary.TypeClass.TYPE_ANYREAL :
        F_IsAnyEqualToUnionValue := FALSE;

    IBaseLibrary.TypeClass.TYPE_LAZY :
        F_IsAnyEqualToUnionValue := FALSE;

    IBaseLibrary.TypeClass.TYPE_LTIME :
        F_IsAnyEqualToUnionValue := uExpectedOrActual.ltimeExpectedOrActual = AnyExpectedOrActual.ltimeExpectedOrActual;

    IBaseLibrary.TypeClass.TYPE_BITCONST :
        F_IsAnyEqualToUnionValue := FALSE;

    IBaseLibrary.TypeClass.TYPE_INTERFACE :
        F_IsAnyEqualToUnionValue := FALSE;

    ELSE
        F_IsAnyEqualToUnionValue := FALSE;
END_CASE

END_FUNCTION

// POUs/Functions/IS_TEST_FINISHED
(* Check if a certain test in the current suite is finished *)
FUNCTION IS_TEST_FINISHED : BOOL
VAR_INPUT
    TestName : Tc2_System.T_MaxString;
END_VAR
VAR
    Counter : UINT;
    CurrentTest : FB_Test;
END_VAR

IS_TEST_FINISHED := FALSE;

FOR Counter := 1 TO GVL_TcUnit.CurrentTestSuiteBeingCalled^.GetNumberOfTests() BY 1 DO
    CurrentTest := GVL_TcUnit.CurrentTestSuiteBeingCalled^.Tests[Counter];
    IF CurrentTest.TestName = TestName THEN
        IS_TEST_FINISHED := CurrentTest.IsFinished();
        RETURN;
    END_IF
END_FOR

END_FUNCTION

// POUs/FB_Test
(*
    This function block holds all data that defines a test.
*)
FUNCTION_BLOCK FB_Test
VAR
    TestName : Tc2_System.T_MaxString; 
    TestIsFinished : BOOL;
    TestIsSkipped : BOOL; // This is set to true, if test is disabled (by putting the string "disabled_" in front of the test name
    NumberOfAssertions : UINT;

    (* Failure parameters. If TestIsFailed is TRUE, the other parameters will hold values as well *)
    TestIsFailed : BOOL; // Indication of whether this test has at least one failed assert
    AssertionMessage : Tc2_System.T_MaxString; // Assertion message for the first assertion in this test
    AssertionType : E_AssertionType; // Assertion type for the first assertion in this test
END_VAR

METHOD PUBLIC GetAssertionMessage : Tc2_System.T_MaxString
GetAssertionMessage := AssertionMessage;
END_METHOD

METHOD PUBLIC GetAssertionType : E_AssertionType
GetAssertionType := AssertionType;
END_METHOD

METHOD PUBLIC GetName : Tc2_System.T_MaxString;
GetName := TestName;
END_METHOD

METHOD PUBLIC GetNumberOfAssertions : UINT
GetNumberOfAssertions := NumberOfAssertions;
END_METHOD

METHOD PUBLIC IsFailed : BOOL
IsFailed := TestIsFailed;
END_METHOD

METHOD PUBLIC IsFinished : BOOL
IsFinished := TestIsFinished;
END_METHOD

METHOD PUBLIC IsSkipped : BOOL
IsSkipped := TestIsSkipped;
END_METHOD

(* Sets the assertion message. If one already exists, it's not overwritten as we keep the first assertion in the test *)
METHOD PUBLIC SetAssertionMessage
VAR_INPUT
    AssertMessage : Tc2_System.T_MaxString;
END_VAR
IF Tc2_Standard.LEN(STR := AssertionMessage) = 0 THEN
    AssertionMessage := AssertMessage;
END_IF
END_METHOD

(* Sets the assertion type. If one already exists, it's not overwritten as we keep the first assertion in the test *)
METHOD PUBLIC SetAssertionType
VAR_INPUT
    AssertType : E_AssertionType;
END_VAR
IF AssertionType = E_AssertionType.Type_UNDEFINED THEN
    AssertionType := AssertType;
END_IF
END_METHOD

METHOD PUBLIC SetFailed
TestIsFailed := TRUE;
END_METHOD

METHOD SetFinished : BOOL
TestIsFinished := TRUE;
END_METHOD

METHOD PUBLIC SetName
VAR_INPUT
    Name : Tc2_System.T_MaxString;
END_VAR
TestName := Name;
END_METHOD

METHOD PUBLIC SetNumberOfAssertions
VAR_INPUT
    NoOfAssertions : UINT;
END_VAR
NumberOfAssertions := NoOfAssertions;
END_METHOD

(* Sets the test case to skipped *)
METHOD PUBLIC SetSkipped
TestIsSkipped := TRUE;
END_METHOD

END_FUNCTION_BLOCK

// POUs/Functions/RUN
(*
    This function runs all test suites that have been initialized.
*)
FUNCTION RUN

GVL_TcUnit.TcUnitRunner.RunTestSuiteTests();

END_FUNCTION

// POUs/Functions/TEST_FINISHED
(* Sets the currently running test as finished *)
FUNCTION TEST_FINISHED : BOOL
VAR
    TestName : Tc2_System.T_MaxString;
    Counter : UINT := 0;
END_VAR

// Grab the currently running test name
TestName := GVL_TcUnit.CurrentTestNameBeingCalled;

TEST_FINISHED := FALSE;
(* Find the test suite and:
   1. Set the test in that test suite as finished
   2. Calculate and set the number of asserts made for that test
*)
FOR Counter := 1 TO GVL_TcUnit.NumberOfInitializedTestSuites BY 1 DO
    IF GVL_TcUnit.TestSuiteAddresses[Counter] = GVL_TcUnit.CurrentTestSuiteBeingCalled THEN
        GVL_TcUnit.TestSuiteAddresses[Counter]^.SetTestFinished(TestName := GVL_TcUnit.CurrentTestNameBeingCalled);
        GVL_TcUnit.TestSuiteAddresses[Counter]^.CalculateAndSetNumberOfAssertsForTest(TestName := GVL_TcUnit.CurrentTestNameBeingCalled);
        GVL_TcUnit.CurrentTestIsFinished := TRUE;
        TEST_FINISHED := TRUE;
        RETURN;
    END_IF
END_FOR

END_FUNCTION

// POUs/Functions/TEST_FINISHED_NAMED
(* Sets a test defined by TestName as finished. Note that the TestName-input must match
   a TestName that has been previously defined in this test suite. *)
FUNCTION TEST_FINISHED_NAMED
VAR_INPUT
    TestName : Tc2_System.T_MaxString;
END_VAR
VAR
    Counter : UINT := 0;
    FoundTestName : BOOL := FALSE;
END_VAR
VAR_STAT
    FailedLookupCounter : UINT := 0;
    AlreadyPrintedFinalWarning : BOOL := FALSE;
END_VAR
VAR CONSTANT
    MaxNumberOfNonExistentTestNamesFailedLookups : UINT := 3;
END_VAR

(* Find the test suite and:
   1. Set the test in that test suite as finished
   2. Calculate and set the number of asserts made for that test
*)
FOR Counter := 1 TO GVL_TcUnit.NumberOfInitializedTestSuites BY 1 DO
    IF GVL_TcUnit.TestSuiteAddresses[Counter] = GVL_TcUnit.CurrentTestSuiteBeingCalled THEN
        FoundTestName := GVL_TcUnit.TestSuiteAddresses[Counter]^.SetTestFinished(TestName := TestName);
        IF NOT FoundTestName THEN
            IF FailedLookupCounter < MaxNumberOfNonExistentTestNamesFailedLookups THEN
                GVL_TcUnit.AdsMessageQueue.WriteLog(MsgCtrlMask := Tc2_System.ADSLOG_MSGTYPE_ERROR,
                                                    MsgFmtStr := 'Failed to find test $'%s$'',
                                                    StrArg := TestName);
                FailedLookupCounter := FailedLookupCounter + 1;
                (* Abort TcUnit *)
                GVL_TcUnit.TcUnitRunner.AbortRunningTestSuiteTests();
            ELSIF NOT AlreadyPrintedFinalWarning THEN
                GVL_TcUnit.AdsMessageQueue.WriteLog(MsgCtrlMask := Tc2_System.ADSLOG_MSGTYPE_ERROR,
                                                    MsgFmtStr := 'Excess failed attempts to mark test finished, failed. Further warnings will be suppressed',
                                                    StrArg := TestName);
                AlreadyPrintedFinalWarning := TRUE;
            END_IF
        ELSE
            GVL_TcUnit.TestSuiteAddresses[Counter]^.CalculateAndSetNumberOfAssertsForTest(TestName := TestName);
            GVL_TcUnit.CurrentTestIsFinished := TRUE;
        END_IF
        RETURN;
    END_IF
END_FOR

END_FUNCTION

// POUs/FB_AdjustAssertFailureMessageToMax253CharLength
(*
    This function block is responsible for making sure that the asserted test instance path and test message are not
    loo long. The total printed message can not be more than 253 characters long.
*)
FUNCTION_BLOCK FB_AdjustAssertFailureMessageToMax253CharLength
VAR_INPUT
    MsgFmtString : Tc2_System.T_MaxString; // Test instance path
    StringArg : Tc2_System.T_MaxString; // Test message
END_VAR
VAR_OUTPUT
    MsgFmtStringProcessed : Tc2_System.T_MaxString;
    StringArgProcessed : Tc2_System.T_MaxString;
END_VAR
VAR
    MsgFmtStringTemp : Tc2_System.T_MaxString;
    TestNameTooLong : STRING := '...TestName too long';
    TestMsgTooLong : STRING := '...TestMsg too long';
END_VAR
VAR CONSTANT
    MSG_FMT_STRING_MAX_NUMBER_OF_CHARACTERS : INT := 253; // This is actually 254, but if StrArg-argument is used (which it is in TcUnit) it is 253.
END_VAR

// Check if any of the two strings are too long (or the combination of them)

// All OK
IF (Tc2_Standard.LEN(STR := MsgFmtString) + LEN(STR := StringArg)) <= MSG_FMT_STRING_MAX_NUMBER_OF_CHARACTERS THEN
    MsgFmtStringProcessed := MsgFmtString;
    StringArgProcessed := StringArg;
// If test instance path is longer than 253 chars, shorten it down to 253 characters and additionally with the length of the '...TestName too long'. Add the text '...TestName too long' to the test instance path. Leave no characters for the message.
ELSIF Tc2_Standard.LEN(STR := MsgFmtString) > MSG_FMT_STRING_MAX_NUMBER_OF_CHARACTERS THEN
    MsgFmtStringTemp := Tc2_Standard.LEFT(STR := MsgFmtString, SIZE := (MSG_FMT_STRING_MAX_NUMBER_OF_CHARACTERS - Tc2_Standard.LEN(STR := TestNameTooLong)));
    MsgFmtStringProcessed := Tc2_Standard.CONCAT(STR1 := MsgFmtStringTemp, STR2 := TestNameTooLong);
    StringArgProcessed := '';
// If test message is too long (so we cant fit the text "...TestMsg too long" to the end of it) , shorten it (so that we can fit the text)
ELSIF (MSG_FMT_STRING_MAX_NUMBER_OF_CHARACTERS - Tc2_Standard.LEN(STR := TestMsgTooLong)) >= Tc2_Standard.LEN(STR := MsgFmtString) THEN
    MsgFmtStringProcessed := MsgFmtString;
    StringArgProcessed := Tc2_Standard.LEFT(STR := StringArg,
                                            SIZE := (MSG_FMT_STRING_MAX_NUMBER_OF_CHARACTERS - Tc2_Standard.LEN(STR := TestMsgTooLong) - Tc2_Standard.LEN(STR := MsgFmtStringProcessed)));
    StringArgProcessed := Tc2_Standard.CONCAT(STR1 := StringArgProcessed, STR2 := TestMsgTooLong);
// If test instance path is too long (length is between 233 and 253 characters long), shorten it and add the text '...TestName too long'. Leave no characters for the message
ELSE
    MsgFmtStringTemp := Tc2_Standard.LEFT(STR := MsgFmtString, SIZE := (MSG_FMT_STRING_MAX_NUMBER_OF_CHARACTERS - Tc2_Standard.LEN(STR := TestNameTooLong)));
    MsgFmtStringProcessed := Tc2_Standard.CONCAT(STR1 := MsgFmtStringTemp, STR2 := TestNameTooLong);
    StringArgProcessed := '';
END_IF

END_FUNCTION_BLOCK

// POUs/FB_AdsAssertMessageFormatter
(*
    This function block is responsible for printing the results of the assertions using the built-in
    ADSLOGSTR functionality provided by the Tc2_System library. This sends the result using ADS, which
    is consumed by the error list of Visual Studio.
*)
FUNCTION_BLOCK FB_AdsAssertMessageFormatter IMPLEMENTS I_AssertMessageFormatter

METHOD LogAssertFailure
VAR_INPUT
    Expected : Tc2_System.T_MaxString;
    Actual : Tc2_System.T_MaxString;
    Message : Tc2_System.T_MaxString;
    TestInstancePath : Tc2_System.T_MaxString;
END_VAR
VAR
    AdjustAssertFailureMessageToMax253CharLength : FB_AdjustAssertFailureMessageToMax253CharLength;
    TestInstancePathCleaned : Tc2_System.T_MaxString;
    TestInstancePathFinal : Tc2_System.T_MaxString;
    ReturnValue : DINT;
    TestInstancePathProcessed : Tc2_System.T_MaxString;
    MessageProcessed : Tc2_System.T_MaxString;
END_VAR
TestInstancePathCleaned := F_RemoveInstancePathAndProjectNameFromTestInstancePath(TestInstancePath);
TestInstancePathFinal := Tc2_Standard.CONCAT(STR1 := 'FAILED TEST $'', STR2 := TestInstancePathCleaned);
TestInstancePathFinal := Tc2_Standard.CONCAT(STR1 := TestInstancePathFinal, STR2 := '$'');

IF Tc2_Standard.LEN(STR := Expected) > 0 THEN
    TestInstancePathFinal := Tc2_Standard.CONCAT(STR1 := TestInstancePathFinal, STR2 := ', EXP: ');
    TestInstancePathFinal := Tc2_Standard.CONCAT(STR1 := TestInstancePathFinal, STR2 := Expected);
END_IF
IF Tc2_Standard.LEN(STR := Actual) > 0 THEN
    TestInstancePathFinal := Tc2_Standard.CONCAT(STR1 := TestInstancePathFinal, STR2 := ', ACT: ');
    TestInstancePathFinal := Tc2_Standard.CONCAT(STR1 := TestInstancePathFinal, STR2 := Actual);
END_IF
IF Tc2_Standard.LEN(STR := Message) > 0 THEN
    TestInstancePathFinal := Tc2_Standard.CONCAT(STR1 := TestInstancePathFinal, STR2 := ', MSG: %s');
END_IF

AdjustAssertFailureMessageToMax253CharLength(MsgFmtString := TestInstancePathFinal,
                                             StringArg := Message,
                                             MsgFmtStringProcessed => TestInstancePathProcessed,
                                             StringArgProcessed => MessageProcessed);

GVL_TcUnit.AdsMessageQueue.WriteLog(MsgCtrlMask := Tc2_System.ADSLOG_MSGTYPE_ERROR,
                                    MsgFmtStr := TestInstancePathProcessed,
                                    StrArg := MessageProcessed);
END_METHOD

END_FUNCTION_BLOCK

// POUs/FB_AdsLogStringMessageFifoQueue
(* This function block is responsible for making sure that the ADSLOGSTR-messages to the ADS-router are transmitted
   cyclically and not in a burst. The reason this is necessary is because that if too many messages are sent at the
   same time some get lost and are never printed to the error list output
*)
FUNCTION_BLOCK FB_AdsLogStringMessageFifoQueue
VAR
    ArrayBuffer : ARRAY[0..((GVL_Param_TcUnit.AdsLogMessageFifoRingBufferSize * (SIZEOF(ST_ADSLogStringMessage) + MEM_RING_BUFFER_INTERNAL_USE_PER_DATA_RECORD)) - 1)] OF BYTE;
    MemRingBuffer : Tc2_Utilities.FB_MemRingBuffer;
    TimerBetweenMessages : Tc2_Standard.TON := (IN := TRUE, PT := TIME_BETWEEN_MESSAGES);
END_VAR
VAR CONSTANT
    MEM_RING_BUFFER_INTERNAL_USE_PER_DATA_RECORD : USINT := 4;
    TIME_BETWEEN_MESSAGES : TIME := T#10MS;
END_VAR
VAR_TEMP
    MessageToBeSent : ST_ADSLogStringMessage;
    ErrorGet : BOOL;
    ReturnValue : DINT;
END_VAR

TimerBetweenMessages();
IF GetLogCount() > 0 THEN
    // Timer has elapsed, print message
    IF TimerBetweenMessages.Q THEN
        GetAndRemoveLogFromQueue(AdsLogStringMessage => MessageToBeSent,
                                 Error => ErrorGet);
        IF NOT ErrorGet THEN
            ReturnValue := Tc2_System.ADSLOGSTR(msgCtrlMask := MessageToBeSent.MsgCtrlMask,
                                                msgFmtStr := MessageToBeSent.MsgFmtStr,
                                                strArg := MessageToBeSent.StrArg);
        END_IF
        TimerBetweenMessages(IN := FALSE); // Reset timer
        TimerBetweenMessages.IN := TRUE;
    END_IF
END_IF

(* Reads and removes the oldest message *)
METHOD PRIVATE GetAndRemoveLogFromQueue
VAR_OUTPUT
    AdsLogStringMessage : ST_ADSLogStringMessage;
    Error : BOOL; // Buffer empty
END_VAR
MemRingBuffer.A_RemoveHead(pRead := ADR(AdsLogStringMessage),
                           cbRead := SIZEOF(ST_ADSLogStringMessage),
                           pBuffer := ADR(ArrayBuffer),
                           cbBuffer := SIZEOF(ArrayBuffer));
Error := NOT MemRingBuffer.bOk;
END_METHOD

METHOD PRIVATE GetLogCount : UDINT
GetLogCount := MemRingBuffer.nCount;
END_METHOD

(* Writes a new data set into the ring buffer *)
METHOD PUBLIC WriteLog
VAR_INPUT
    MsgCtrlMask : DWORD;
    MsgFmtStr : Tc2_System.T_MaxString;
    StrArg : Tc2_System.T_MaxString;
END_VAR
VAR_OUTPUT
    Error : BOOL; // Buffer overflow
END_VAR
VAR
    AdsLogStringMessage : ST_AdsLogStringMessage;
END_VAR
(* Only log message types of ERROR if log extended results is not enabled *)
IF MsgCtrlMask = Tc2_System.ADSLOG_MSGTYPE_ERROR OR GVL_Param_TcUnit.LogExtendedResults THEN
    AdsLogStringMessage.MsgCtrlMask := MsgCtrlMask;
    AdsLogStringMessage.MsgFmtStr := MsgFmtStr;
    AdsLogStringMessage.StrArg := StrArg;

    MemRingBuffer.A_AddTail(pWrite := ADR(AdsLogStringMessage),
                            cbWrite := SIZEOF(ST_AdsLogStringMessage),
                            pBuffer := ADR(ArrayBuffer),
                            cbBuffer := SIZEOF(ArrayBuffer));

    Error := NOT MemRingBuffer.bOk;
END_IF
END_METHOD

END_FUNCTION_BLOCK

// POUs/FB_AdsTestResultLogger
(*
    This function block reports the results from the tests using the built-in ADSLOGSTR functionality
    provided by the Tc2_System library. This sends the result using ADS, which is consumed by the "Error List"
    of Visual Studio (which can print Errors, Warnings and Messages).
*)
FUNCTION_BLOCK FB_AdsTestResultLogger IMPLEMENTS I_TestResultLogger
VAR
    TestResults : I_TestResults;

    PrintingTestSuiteResultNumber : UINT(1..GVL_Param_TcUnit.MaxNumberOfTestSuites);
    PrintingTestSuiteTrigger : Tc2_Standard.R_TRIG;

    (* This flag is set once the final end result has printed *)
    PrintedFinalTestResults : BOOL;

    (* This flag is set once the test suites result have been printed *)
    PrintedTestSuitesResults : BOOL;
END_VAR

METHOD FB_init : BOOL
VAR_INPUT
	bInitRetains : BOOL; // if TRUE, the retain variables are initialized (warm start / cold start)
	bInCopyCode : BOOL;  // if TRUE, the instance afterwards gets moved into the copy code (online change)
    iTestResults : I_TestResults;
END_VAR
TestResults := iTestResults;
END_METHOD

METHOD PUBLIC LogTestSuiteResults
VAR
    TcUnitTestResults : REFERENCE TO ST_TestSuiteResults;
    StringToPrint : Tc2_System.T_MaxString; 
    TestsInTestSuiteCounter : UINT(1..GVL_Param_TcUnit.MaxNumberOfTestsForEachTestSuite);
END_VAR
VAR CONSTANT
    TEST_STATUS_SKIP : STRING := 'SKIP';
    TEST_STATUS_PASS : STRING := 'PASS';
    TEST_STATUS_FAIL : STRING := 'FAIL';
END_VAR
TcUnitTestResults REF= TestResults.GetTestSuiteResults();

IF PrintingTestSuiteResultNumber <= GVL_TcUnit.NumberOfInitializedTestSuites AND NOT PrintedTestSuitesResults THEN
    
    PrintingTestSuiteTrigger(CLK := GVL_TcUnit.TestSuiteAddresses[PrintingTestSuiteResultNumber]^.AreAllTestsFinished());
    IF PrintingTestSuiteTrigger.Q THEN
        StringToPrint := Tc2_Standard.CONCAT(STR1 := '| Test suite ID=',
                                             STR2 := UINT_TO_STRING(TcUnitTestResults.TestSuiteResults[PrintingTestSuiteResultNumber].Identity));
        StringToPrint := Tc2_Standard.CONCAT(STR1 := StringToPrint,
                                             STR2 :=  ' $'%s$'');

        (* Print test suite name and ID *)
        GVL_TcUnit.AdsMessageQueue.WriteLog(MsgCtrlMask := Tc2_System.ADSLOG_MSGTYPE_HINT,
                                            MsgFmtStr := StringToPrint,
                                            StrArg := TcUnitTestResults.TestSuiteResults[PrintingTestSuiteResultNumber].Name);

        (* Print number of tests/number of failed tests in test suite *)
        StringToPrint := Tc2_Standard.CONCAT(STR1 := '| ID=',
                                             STR2 := UINT_TO_STRING(TcUnitTestResults.TestSuiteResults[PrintingTestSuiteResultNumber].Identity));
        StringToPrint := Tc2_Standard.CONCAT(STR1 := StringToPrint,
                                             STR2 := ' number of tests=');
        StringToPrint := Tc2_Standard.CONCAT(STR1 := StringToPrint,
                                             STR2 := UINT_TO_STRING(TcUnitTestResults.TestSuiteResults[PrintingTestSuiteResultNumber].NumberOfTests));
        StringToPrint := Tc2_Standard.CONCAT(STR1 := StringToPrint,
                                             STR2 := ', number of failed tests=');
        StringToPrint := Tc2_Standard.CONCAT(STR1 := StringToPrint,
                                             STR2 := UINT_TO_STRING(TcUnitTestResults.TestSuiteResults[PrintingTestSuiteResultNumber].NumberOfFailedTests));

        GVL_TcUnit.AdsMessageQueue.WriteLog(MsgCtrlMask := Tc2_System.ADSLOG_MSGTYPE_HINT,
                                            MsgFmtStr := StringToPrint,
                                            StrArg := '');

        (* Iterate and print all tests in test suite *)
        FOR TestsInTestSuiteCounter := 1 TO TcUnitTestResults.TestSuiteResults[PrintingTestSuiteResultNumber].NumberOfTests BY 1 DO
            (* Print test name *)
            GVL_TcUnit.AdsMessageQueue.WriteLog(MsgCtrlMask := Tc2_System.ADSLOG_MSGTYPE_HINT,
                                                MsgFmtStr := '| Test name=%s',
                                                StrArg := TcUnitTestResults.TestSuiteResults[PrintingTestSuiteResultNumber].TestCaseResults[TestsInTestSuiteCounter].TestName);
            (* Print test class name *)
            GVL_TcUnit.AdsMessageQueue.WriteLog(MsgCtrlMask := Tc2_System.ADSLOG_MSGTYPE_HINT,
                                                MsgFmtStr := '| Test class name=%s',
                                                StrArg := TcUnitTestResults.TestSuiteResults[PrintingTestSuiteResultNumber].TestCaseResults[TestsInTestSuiteCounter].TestClassName);

            (* Print test result/status (SUCCESS, FAILED, SKIPPED) + number of assertions made *)
            IF TcUnitTestResults.TestSuiteResults[PrintingTestSuiteResultNumber].TestCaseResults[TestsInTestSuiteCounter].TestIsFailed THEN
                StringToPrint := Tc2_Standard.CONCAT(STR1 := '| Test status=', STR2 := TEST_STATUS_FAIL);
            ELSIF TcUnitTestResults.TestSuiteResults[PrintingTestSuiteResultNumber].TestCaseResults[TestsInTestSuiteCounter].TestIsSkipped THEN
                StringToPrint := Tc2_Standard.CONCAT(STR1 := '| Test status=', STR2 := TEST_STATUS_SKIP);
            ELSE
                StringToPrint := Tc2_Standard.CONCAT(STR1 := '| Test status=', STR2 := TEST_STATUS_PASS);
			END_IF

            StringToPrint := Tc2_Standard.CONCAT(STR1 := StringToPrint, STR2 := ', number of asserts=');
            StringToPrint := Tc2_Standard.CONCAT(STR1 := StringToPrint, STR2 :=
                                                 UINT_TO_STRING(TcUnitTestResults.TestSuiteResults[PrintingTestSuiteResultNumber].TestCaseResults[TestsInTestSuiteCounter].NumberOfAsserts));
            GVL_TcUnit.AdsMessageQueue.WriteLog(MsgCtrlMask := Tc2_System.ADSLOG_MSGTYPE_HINT,
                                                MsgFmtStr := StringToPrint,
                                                StrArg := '');

            (* Print assertion/failure message (if existing) *)
            IF (Tc2_Standard.LEN(STR := TcUnitTestResults.TestSuiteResults[PrintingTestSuiteResultNumber].TestCaseResults[TestsInTestSuiteCounter].FailureMessage) > 0) THEN
                GVL_TcUnit.AdsMessageQueue.WriteLog(MsgCtrlMask := Tc2_System.ADSLOG_MSGTYPE_HINT,
                                                    MsgFmtStr := '| Test assert message=%s',
                                                    StrArg := TcUnitTestResults.TestSuiteResults[PrintingTestSuiteResultNumber].TestCaseResults[TestsInTestSuiteCounter].FailureMessage);
            END_IF

            (* Print assertion/failure type (if existing) *)
            IF TcUnitTestResults.TestSuiteResults[PrintingTestSuiteResultNumber].TestCaseResults[TestsInTestSuiteCounter].FailureType <> E_AssertionType.Type_UNDEFINED THEN
                GVL_TcUnit.AdsMessageQueue.WriteLog(MsgCtrlMask := Tc2_System.ADSLOG_MSGTYPE_HINT,
                                                    MsgFmtStr := '| Test assert type=%s',
                                                    StrArg := F_AssertionTypeToString(AssertionType :=
                                                        TcUnitTestResults.TestSuiteResults[PrintingTestSuiteResultNumber].TestCaseResults[TestsInTestSuiteCounter].FailureType));
            END_IF

		END_FOR

        IF PrintingTestSuiteResultNumber = GVL_TcUnit.NumberOfInitializedTestSuites THEN
            PrintedTestSuitesResults := TRUE;
        ELSE
            PrintingTestSuiteResultNumber := PrintingTestSuiteResultNumber + 1;
        END_IF
        PrintingTestSuiteTrigger(CLK := FALSE); // Reset trigger
    END_IF
END_IF

(* Log end results once all test suites have finished running *)
IF (GVL_TcUnit.NumberOfInitializedTestSuites = 0 OR PrintingTestSuiteResultNumber = GVL_TcUnit.NumberOfInitializedTestSuites)
    AND NOT PrintedFinalTestResults AND TestResults.GetAreTestResultsAvailable() THEN
    GVL_TcUnit.AdsMessageQueue.WriteLog(MsgCtrlMask := Tc2_System.ADSLOG_MSGTYPE_ERROR,
                                        MsgFmtStr := '%s',
                                        StrArg := '| ==========TESTS FINISHED RUNNING==========');
    GVL_TcUnit.AdsMessageQueue.WriteLog(MsgCtrlMask := Tc2_System.ADSLOG_MSGTYPE_ERROR,
                                        MsgFmtStr := '| Test suites: %s',
                                        StrArg := UINT_TO_STRING(TcUnitTestResults.NumberOfTestSuites));
    GVL_TcUnit.AdsMessageQueue.WriteLog(MsgCtrlMask := Tc2_System.ADSLOG_MSGTYPE_ERROR,
                                        MsgFmtStr := '| Tests: %s',
                                        StrArg := UINT_TO_STRING(TcUnitTestResults.NumberOfTestCases));
    GVL_TcUnit.AdsMessageQueue.WriteLog(MsgCtrlMask := Tc2_System.ADSLOG_MSGTYPE_ERROR,
                                        MsgFmtStr := '| Successful tests: %s',
                                        StrArg := UINT_TO_STRING(TcUnitTestResults.NumberOfSuccessfulTestCases));
    GVL_TcUnit.AdsMessageQueue.WriteLog(MsgCtrlMask := Tc2_System.ADSLOG_MSGTYPE_ERROR,
                                        MsgFmtStr := '| Failed tests: %s',
                                        StrArg := UINT_TO_STRING(TcUnitTestResults.NumberOfFailedTestCases));
    GVL_TcUnit.AdsMessageQueue.WriteLog(MsgCtrlMask := Tc2_System.ADSLOG_MSGTYPE_ERROR,
                                        MsgFmtStr := '%s',
                                        StrArg := '| ======================================');
    PrintedFinalTestResults := TRUE;
END_IF
END_METHOD

END_FUNCTION_BLOCK

// POUs/FB_AssertArrayResultStatic
(*
    This function block is responsible for keeping track of which array-asserts that have been made.
    The reason we need to keep track of these is because if the user does the same assert twice
    (because of running a test suite over several PLC-cycles) we want to know it so we don't print several times
    (if the assert fails). An instance of an array-assert is keyed/identified with the following parameters as key:
    - Array-size (in bytes) of the expecteds
    - Datatype of the expecteds
    - Array-size (in bytes) of the actuals
    - Datatype of the actuals
    - Message (string)
    - Test instance path (string)
*)
FUNCTION_BLOCK FB_AssertArrayResultStatic
VAR
    (* The total number of instances of each of the "AssertArrayResults" *)
    AssertArrayResults : ARRAY[1..GVL_Param_TcUnit.MaxNumberOfAssertsForEachTestSuite] OF ST_AssertArrayResult;

    (* The total number of unique asserts *)
    TotalArrayAsserts : UINT := 0;

    (* Function block to get the current task cycle *)
    GetCurrentTaskIndex : Tc2_System.GETCURTASKINDEX;

    (* The total number of instances of each of the "AssertArrayResults" *)
    AssertArrayResultInstances : ARRAY[1..GVL_Param_TcUnit.MaxNumberOfAssertsForEachTestSuite] OF ST_AssertArrayResultInstances;

    (* The last PLC cycle count *)
    CycleCount : UDINT;

    (* Only run first cycle *)
    FirstCycleExecuted : BOOL;
END_VAR

METHOD PRIVATE AddAssertArrayResult
VAR_INPUT
    ExpectedsSize : UDINT;
    ExpectedsTypeClass : IBaseLibrary.TypeClass;
    ActualsSize : UDINT;
    ActualsTypeClass : IBaseLibrary.TypeClass;
    Message : Tc2_System.T_MaxString;
    TestInstancePath : Tc2_System.T_MaxString;
END_VAR
TotalArrayAsserts := TotalArrayAsserts + 1;
AssertArrayResults[TotalArrayAsserts].ExpectedsSize := ExpectedsSize;
AssertArrayResults[TotalArrayAsserts].ExpectedsTypeClass := ExpectedsTypeClass;
AssertArrayResults[TotalArrayAsserts].ActualsSize := ActualsSize;
AssertArrayResults[TotalArrayAsserts].ActualsTypeClass := ActualsTypeClass;
AssertArrayResults[TotalArrayAsserts].Message := Message;
AssertArrayResults[TotalArrayAsserts].TestInstancePath := TestInstancePath;
END_METHOD

METHOD PRIVATE CopyDetectionCountAndResetDetectionCountInThisCycle
VAR
    IteratorCounter : UINT;
END_VAR
FOR IteratorCounter := 1 TO GVL_Param_TcUnit.MaxNumberOfAssertsForEachTestSuite BY 1 DO
    AssertArrayResultInstances[IteratorCounter].DetectionCount := AssertArrayResultInstances[IteratorCounter].DetectionCountThisCycle;
    AssertArrayResultInstances[IteratorCounter].DetectionCountThisCycle := 0;
END_FOR
END_METHOD

METHOD PRIVATE CreateAssertResultInstance
VAR_INPUT
    ExpectedsSize : UDINT;
    ExpectedsTypeClass : IBaseLibrary.TypeClass;
    ActualsSize : UDINT;
    ActualsTypeClass : IBaseLibrary.TypeClass;
    Message : Tc2_System.T_MaxString;
    TestInstancePath : Tc2_System.T_MaxString;
END_VAR
VAR
    IteratorCounter : UINT;
END_VAR
FOR IteratorCounter := 1 TO GVL_Param_TcUnit.MaxNumberOfAssertsForEachTestSuite BY 1 DO
    IF AssertArrayResultInstances[IteratorCounter].DetectionCount = 0 AND
        AssertArrayResultInstances[IteratorCounter].DetectionCountThisCycle = 0 THEN // Find first free spot
        AssertArrayResultInstances[IteratorCounter].AssertArrayResult.ExpectedsSize := ExpectedsSize;
        AssertArrayResultInstances[IteratorCounter].AssertArrayResult.ExpectedsTypeClass := ExpectedsTypeClass;
        AssertArrayResultInstances[IteratorCounter].AssertArrayResult.ActualsSize := ActualsSize;
        AssertArrayResultInstances[IteratorCounter].AssertArrayResult.ActualsTypeClass := ActualsTypeClass;
        AssertArrayResultInstances[IteratorCounter].AssertArrayResult.Message := Message;
        AssertArrayResultInstances[IteratorCounter].AssertArrayResult.TestInstancePath := TestInstancePath;
        AssertArrayResultInstances[IteratorCounter].DetectionCountThisCycle := 1;
        EXIT;
    END_IF
END_FOR
END_METHOD

METHOD PRIVATE GetDetectionCount : UINT
VAR_INPUT
    ExpectedsSize : UDINT;
    ExpectedsTypeClass : IBaseLibrary.TypeClass;
    ActualsSize : UDINT;
    ActualsTypeClass : IBaseLibrary.TypeClass;
    Message : Tc2_System.T_MaxString;
    TestInstancePath : Tc2_System.T_MaxString;
END_VAR
VAR
    IteratorCounter : UINT;
END_VAR
FOR IteratorCounter := 1 TO GVL_Param_TcUnit.MaxNumberOfAssertsForEachTestSuite BY 1 DO
    IF AssertArrayResultInstances[IteratorCounter].AssertArrayResult.ExpectedsSize = ExpectedsSize AND
       AssertArrayResultInstances[IteratorCounter].AssertArrayResult.ExpectedsTypeClass = ExpectedsTypeClass AND
       AssertArrayResultInstances[IteratorCounter].AssertArrayResult.ActualsSize = ActualsSize AND
       AssertArrayResultInstances[IteratorCounter].AssertArrayResult.ActualsTypeClass = ActualsTypeClass AND
       AssertArrayResultInstances[IteratorCounter].AssertArrayResult.Message = Message AND
       AssertArrayResultInstances[IteratorCounter].AssertArrayResult.TestInstancePath = TestInstancePath THEN
        GetDetectionCount := AssertArrayResultInstances[IteratorCounter].DetectionCount;
    END_IF
END_FOR
END_METHOD

METHOD PRIVATE GetDetectionCountThisCycle : UINT
VAR_INPUT
    ExpectedsSize : UDINT;
    ExpectedsTypeClass : IBaseLibrary.TypeClass;
    ActualsSize : UDINT;
    ActualsTypeClass : IBaseLibrary.TypeClass;
    Message : Tc2_System.T_MaxString;
    TestInstancePath : Tc2_System.T_MaxString;
END_VAR
VAR
    IteratorCounter : UINT;
END_VAR
FOR IteratorCounter := 1 TO GVL_Param_TcUnit.MaxNumberOfAssertsForEachTestSuite BY 1 DO
    IF AssertArrayResultInstances[IteratorCounter].AssertArrayResult.ExpectedsSize = ExpectedsSize AND
       AssertArrayResultInstances[IteratorCounter].AssertArrayResult.ExpectedsTypeClass = ExpectedsTypeClass AND
       AssertArrayResultInstances[IteratorCounter].AssertArrayResult.ActualsSize = ActualsSize AND
       AssertArrayResultInstances[IteratorCounter].AssertArrayResult.ActualsTypeClass = ActualsTypeClass AND
       AssertArrayResultInstances[IteratorCounter].AssertArrayResult.Message = Message AND
       AssertArrayResultInstances[IteratorCounter].AssertArrayResult.TestInstancePath = TestInstancePath THEN

        GetDetectionCountThisCycle := AssertArrayResultInstances[IteratorCounter].DetectionCountThisCycle;
    END_IF
END_FOR
END_METHOD

METHOD PUBLIC GetNumberOfArrayAssertsForTest : UINT
VAR_INPUT
    CompleteTestInstancePath : Tc2_System.T_MaxString;
END_VAR
VAR
    Counter : UINT;
    NumberOfArrayAsserts : UINT := 0;
END_VAR
IF TotalArrayAsserts > 0 THEN
    FOR Counter := 1 TO TotalArrayAsserts BY 1 DO
        IF AssertArrayResults[Counter].TestInstancePath = CompleteTestInstancePath THEN
            NumberOfArrayAsserts := NumberOfArrayAsserts + 1;
        END_IF
    END_FOR
END_IF

GetNumberOfArrayAssertsForTest := NumberOfArrayAsserts;
END_METHOD

(*
    This method is called in every assert and returns whether this particular assert has already been called.
    The reason one would like to know whether this assert has already been reported or not is to not report it several
    times to any logging service. Because a test-suite can consist of several tests, and certain tests can require the
    test to run over several cycles it means that certain asserts could be called several times and thus we need to
    keep track of which asserts we've already reported. The user of the framework should not need to care for any of
    this and he/she should be able to call the asserts in any way they find suitable.

    To know what assert this is we need to check for the total combination of:
    - Test message
    - Test instance path
    - Expecteds size (in bytes)
    - Actuals size (in bytes)
    - Expecteds datatype
    - Actuals datatype
    Theoretically we can have a situation where a test has three different asserts, each and one with the same test
    message/test instance path/actuals size&datatype/expecteds size&datatype but called within the same or different
    cycles. In order for us to handle all situations we need a simple algorithm that works according to:
    - Keep track of how many instances the combination of test message/test instance path/expecteds size&datatype/
      actuals size&datatype we have. So for example, if we have called
      Assert(Exp := [5,4,3], Act := [5,4,3], 'Hello there', 'PRG.InstanceTestSuite.Test')
      two times in one cycle, we have two instances of that combination. This is done according to:
    - Iterate all existing reports.
      - If we have a new PLC-cycle, set the current detection-count to zero.
      - If new report does not match in any of the above fields, create it (together with current PLC-cycle).
        Also store the information that we have one instance of this combination and +1 on the detection-count.
      - If new report matches in all of the above, +1 in the detection-count. If this detection-count is larger than
        the stored detection-count for this combination, create a new report and add +1 to the storage of
        the detection-count.
*)
METHOD PUBLIC ReportResult
VAR_INPUT
    ExpectedsSize : UDINT;
    ExpectedsTypeClass : IBaseLibrary.TypeClass;
    ActualsSize : UDINT;
    ActualsTypeClass : IBaseLibrary.TypeClass;
    Message : Tc2_System.T_MaxString;
    TestInstancePath : Tc2_System.T_MaxString;
END_VAR
VAR_OUTPUT
    AlreadyReported : BOOL := FALSE;
END_VAR
VAR
    LocationIndex : UINT;
    DataTypesNotEquals : BOOL;
    DataSizeNotEquals : BOOL;
    DataContentNotEquals : BOOL;
    CurrentCycleCount : UDINT;
    IteratorCounter : UINT;
    DetectionCountTemp : UINT := 0;
    FoundOne : BOOL;
    AdditionalIdenticalAssert : BOOL;
END_VAR
IF NOT FirstCycleExecuted THEN
    GetCurrentTaskIndex();
    FirstCycleExecuted := TRUE;
END_IF

CurrentCycleCount := TwinCAT_SystemInfoVarList._TaskInfo[GetCurrentTaskIndex.index].CycleCount;
(* Is current cycle the same as the last call to this method?
   If not, reset the detection count *)
IF CurrentCycleCount <> CycleCount THEN
    CopyDetectionCountAndResetDetectionCountInThisCycle();
END_IF

FOR IteratorCounter := 1 TO TotalArrayAsserts BY 1 DO
    IF AssertArrayResultInstances[IteratorCounter].AssertArrayResult.ExpectedsSize = ExpectedsSize AND
        AssertArrayResultInstances[IteratorCounter].AssertArrayResult.ExpectedsTypeClass = ExpectedsTypeClass AND
        AssertArrayResultInstances[IteratorCounter].AssertArrayResult.ActualsSize = ActualsSize AND
        AssertArrayResultInstances[IteratorCounter].AssertArrayResult.ActualsTypeClass = ActualsTypeClass AND
        AssertArrayResultInstances[IteratorCounter].AssertArrayResult.Message = Message AND
        AssertArrayResultInstances[IteratorCounter].AssertArrayResult.TestInstancePath = TestInstancePath THEN
        AssertArrayResultInstances[IteratorCounter].DetectionCountThisCycle :=
            AssertArrayResultInstances[IteratorCounter].DetectionCountThisCycle + 1;
            FoundOne := TRUE;
        IF AssertArrayResultInstances[IteratorCounter].DetectionCountThisCycle >
                AssertArrayResultInstances[IteratorCounter].DetectionCount THEN // This assert is new
                AdditionalIdenticalAssert := TRUE;
        END_IF
        EXIT;
    END_IF
END_FOR

(* If not found anything, create the first *)
IF NOT FoundOne THEN
    (* No existing match found, create a new entry *)
    AddAssertArrayResult(ExpectedsSize, ExpectedsTypeClass, ActualsSize, ActualsTypeClass, Message, TestInstancePath);
    CreateAssertResultInstance(ExpectedsSize, ExpectedsTypeClass, ActualsSize, ActualsTypeClass,
                               Message, TestInstancePath);
(* An additional instance of this assert needs to be created *)
ELSIF AdditionalIdenticalAssert THEN
    AddAssertArrayResult(ExpectedsSize, ExpectedsTypeClass, ActualsSize, ActualsTypeClass, Message, TestInstancePath);
(* In all other cases, this assert has already been reported, we don't need to do anything *)
ELSE
    AlreadyReported := TRUE;
END_IF

(* Update the cycle count *)
CycleCount := TwinCAT_SystemInfoVarList._TaskInfo[GetCurrentTaskIndex.index].CycleCount;
END_METHOD

END_FUNCTION_BLOCK

// POUs/FB_AssertResultStatic
(*
    This function block is responsible for keeping track of which asserts that have been made. The reason we need to
    keep track of these is because if the user does the same assert twice (because of running a test suite over several
    PLC-cycles) we want to know it so we don't print several times (if the assert fails).
    An instance of an assert is keyed/identified with the following parameters as key:
    - Value of expected
    - Value of actual
    - Message (string)
    - Test instance path (string)
*)
FUNCTION_BLOCK FB_AssertResultStatic
VAR
    (* The total number of instances of each of the "AssertResults" *)
    AssertResults : ARRAY[1..GVL_Param_TcUnit.MaxNumberOfAssertsForEachTestSuite] OF ST_AssertResult;

    (* The total number of unique asserts *)
    TotalAsserts : UINT := 0;

    (* Function block to get the current task cycle *)
    GetCurrentTaskIndex : Tc2_System.GETCURTASKINDEX;

    (* The total number of instances of each of the "AssertResults" *)
    AssertResultInstances : ARRAY[1..GVL_Param_TcUnit.MaxNumberOfAssertsForEachTestSuite] OF ST_AssertResultInstances;

    (* The last PLC cycle count *)
    CycleCount : UDINT;

    (* Only run first cycle *)
    FirstCycleExecuted : BOOL;
END_VAR

METHOD PRIVATE AddAssertResult
VAR_INPUT
    ExpectedSize : UDINT;
    ExpectedTypeClass : IBaseLibrary.TypeClass;
    ExpectedValue : POINTER TO BYTE;
    ActualSize : UDINT;
    ActualTypeClass : IBaseLibrary.TypeClass;
    ActualValue : POINTER TO BYTE;
    Message : Tc2_System.T_MaxString;
    TestInstancePath : Tc2_System.T_MaxString;
END_VAR
TotalAsserts := TotalAsserts + 1;
AssertResults[TotalAsserts].Expected := F_AnyToUnionValue(AnySize := ExpectedSize, AnyTypeClass := ExpectedTypeClass, AnyValue := ExpectedValue);
AssertResults[TotalAsserts].Actual := F_AnyToUnionValue(AnySize := ActualSize, AnyTypeClass := ActualTypeClass, AnyValue := ActualValue);
AssertResults[TotalAsserts].Message := Message;
AssertResults[TotalAsserts].TestInstancePath := TestInstancePath;
END_METHOD

METHOD PRIVATE CopyDetectionCountAndResetDetectionCountInThisCycle
VAR
    IteratorCounter : UINT;
END_VAR
FOR IteratorCounter := 1 TO GVL_Param_TcUnit.MaxNumberOfAssertsForEachTestSuite BY 1 DO
    AssertResultInstances[IteratorCounter].DetectionCount := AssertResultInstances[IteratorCounter].DetectionCountThisCycle;
    AssertResultInstances[IteratorCounter].DetectionCountThisCycle := 0;
END_FOR
END_METHOD

METHOD PRIVATE CreateAssertResultInstance
VAR_INPUT
    ExpectedSize : UDINT;
    ExpectedTypeClass : IBaseLibrary.TypeClass;
    ExpectedValue : POINTER TO BYTE;
    ActualSize : UDINT;
    ActualTypeClass : IBaseLibrary.TypeClass;
    ActualValue : POINTER TO BYTE;
    Message : Tc2_System.T_MaxString;
    TestInstancePath : Tc2_System.T_MaxString;
END_VAR
VAR
    IteratorCounter : UINT;
END_VAR
FOR IteratorCounter := 1 TO GVL_Param_TcUnit.MaxNumberOfAssertsForEachTestSuite BY 1 DO
    IF AssertResultInstances[IteratorCounter].DetectionCount = 0 AND
        AssertResultInstances[IteratorCounter].DetectionCountThisCycle = 0 THEN // Find first free spot
        AssertResultInstances[IteratorCounter].AssertResult.Expected := F_AnyToUnionValue(AnySize := ExpectedSize, AnyTypeClass := ExpectedTypeClass, AnyValue := ExpectedValue);
        AssertResultInstances[IteratorCounter].AssertResult.Actual := F_AnyToUnionValue(AnySize := ActualSize, AnyTypeClass := ActualTypeClass, AnyValue := ActualValue);
        AssertResultInstances[IteratorCounter].AssertResult.Message := Message;
        AssertResultInstances[IteratorCounter].AssertResult.TestInstancePath := TestInstancePath;
        AssertResultInstances[IteratorCounter].DetectionCountThisCycle := 1;
        EXIT;
    END_IF
END_FOR
END_METHOD

METHOD PRIVATE GetDetectionCount : UINT
VAR_INPUT
    ExpectedSize : UDINT;
    ExpectedTypeClass : IBaseLibrary.TypeClass;
    ExpectedValue : POINTER TO BYTE;
    ActualSize : UDINT;
    ActualTypeClass : IBaseLibrary.TypeClass;
    ActualValue : POINTER TO BYTE;
    Message : Tc2_System.T_MaxString;
    TestInstancePath : Tc2_System.T_MaxString;
END_VAR
VAR
    IteratorCounter : UINT;
END_VAR
FOR IteratorCounter := 1 TO GVL_Param_TcUnit.MaxNumberOfAssertsForEachTestSuite BY 1 DO
    IF F_IsAnyEqualToUnionValue(uExpectedOrActual := AssertResultInstances[IteratorCounter].AssertResult.Expected,
                                 ExpectedOrActualSize := ExpectedSize,
                                 ExpectedOrActualTypeClass := ExpectedTypeClass,
                                 ExpectedOrActualValue := ExpectedValue) AND   
       F_IsAnyEqualToUnionValue(uExpectedOrActual := AssertResultInstances[IteratorCounter].AssertResult.Actual,
                                ExpectedOrActualSize := ActualSize,
                                ExpectedOrActualTypeClass := ActualTypeClass,
                                ExpectedOrActualValue := ActualValue) AND 
        AssertResultInstances[IteratorCounter].AssertResult.Message = Message AND
        AssertResultInstances[IteratorCounter].AssertResult.TestInstancePath = TestInstancePath THEN
        GetDetectionCount := AssertResultInstances[IteratorCounter].DetectionCount;
    END_IF
END_FOR
END_METHOD

METHOD PRIVATE GetDetectionCountThisCycle : UINT
VAR_INPUT
    ExpectedSize : UDINT;
    ExpectedTypeClass : IBaseLibrary.TypeClass;
    ExpectedValue : POINTER TO BYTE;
    ActualSize : UDINT;
    ActualTypeClass : IBaseLibrary.TypeClass;
    ActualValue : POINTER TO BYTE;
    Message : Tc2_System.T_MaxString;
    TestInstancePath : Tc2_System.T_MaxString;
END_VAR
VAR
    IteratorCounter : UINT;
END_VAR
FOR IteratorCounter := 1 TO GVL_Param_TcUnit.MaxNumberOfAssertsForEachTestSuite BY 1 DO
    IF F_IsAnyEqualToUnionValue(uExpectedOrActual := AssertResultInstances[IteratorCounter].AssertResult.Expected,
                                ExpectedOrActualSize := ExpectedSize,
                                ExpectedOrActualTypeClass := ExpectedTypeClass,
                                ExpectedOrActualValue := ExpectedValue) AND   
       F_IsAnyEqualToUnionValue(uExpectedOrActual := AssertResultInstances[IteratorCounter].AssertResult.Actual,
                                ExpectedOrActualSize := ActualSize,
                                ExpectedOrActualTypeClass := ActualTypeClass,
                                ExpectedOrActualValue := ActualValue) AND 
        AssertResultInstances[IteratorCounter].AssertResult.Message = Message AND
        AssertResultInstances[IteratorCounter].AssertResult.Message = TestInstancePath THEN
        GetDetectionCountThisCycle := AssertResultInstances[IteratorCounter].DetectionCountThisCycle;
    END_IF
END_FOR
END_METHOD

METHOD PUBLIC GetNumberOfAssertsForTest : UINT
VAR_INPUT
    CompleteTestInstancePath : Tc2_System.T_MaxString;
END_VAR
VAR
    Counter : UINT;
    NumberOfAsserts : UINT := 0;
END_VAR
IF TotalAsserts > 0 THEN
    FOR Counter := 1 TO TotalAsserts BY 1 DO
        IF AssertResults[Counter].TestInstancePath = CompleteTestInstancePath THEN
            NumberOfAsserts := NumberOfAsserts + 1;
        END_IF
    END_FOR
END_IF

GetNumberOfAssertsForTest := NumberOfAsserts;
END_METHOD

(*
    This method is called in every assert and returns whether this particular assert has already been called.
    The reason one would like to know whether this assert has already been reported or not is to not report it several
    times to any logging service. Because a test-suite can consist of several tests, and certain tests can require the
    test to run over several cycles it means that certain asserts could be called several times and thus we need to
    keep track of which asserts we've already reported. The user of the framework should not need to care for any of
    this and he/she should be able to call the asserts in any way they find suitable.

    To know what assert this is we need to check for the total combination of:
    - Test message
    - Test instance path
    - Expected value
    - Actual value
    Theoretically we can have a situation where a test has three different asserts, each and one with the same test
    message/test instance path/actual value/expected value but called within the same or different cycles. In order for
    us to handle all situations we need a simple algorithm that works according to:
    - Keep track of how many instances the combination of test message/test instance path/expected value/actual value
      we have. So for example, if we have called Assert(Exp := 5, Act := 5, 'Hello there', 'PRG.InstanceTestSuite.Test')
      two times in one cycle, we have two instances of that combination. This is done according to:
    - Iterate all existing reports.
      - If we have a new PLC-cycle, set the current detection-count to zero.
      - If new report does not match in any of the above fields, create it (together with current PLC-cycle).
        Also store the information that we have one instance of this combination and +1 on the detection-count.
      - If new report matches in all of the above, +1 in the detection-count. If this detection-count is larger than
        the stored detection-count for this combination, create a new report and add +1 to the storage of
        the detection-count.
*)
METHOD PUBLIC ReportResult
VAR_INPUT
    ExpectedSize : UDINT;
    ExpectedTypeClass : IBaseLibrary.TypeClass;
    ExpectedValue : POINTER TO BYTE;
    ActualSize : UDINT;
    ActualTypeClass : IBaseLibrary.TypeClass;
    ActualValue : POINTER TO BYTE;
    Message : Tc2_System.T_MaxString;
    TestInstancePath : Tc2_System.T_MaxString;
END_VAR
VAR_OUTPUT
    AlreadyReported : BOOL := FALSE;
END_VAR
VAR
    LocationIndex : UINT;
    DataTypesNotEquals : BOOL;
    DataSizeNotEquals : BOOL;
    DataContentNotEquals : BOOL;
    CurrentCycleCount : UDINT;
    IteratorCounter : UINT;
    DetectionCountTemp : UINT := 0;
    FoundOne : BOOL;
    AdditionalIdenticalAssert : BOOL;
END_VAR
IF NOT FirstCycleExecuted THEN
    GetCurrentTaskIndex();
    FirstCycleExecuted := TRUE;
END_IF

CurrentCycleCount := TwinCAT_SystemInfoVarList._TaskInfo[GetCurrentTaskIndex.index].CycleCount;
(* Is current cycle the same as the last call to this method?
   If not, reset the detection count *)
IF CurrentCycleCount <> CycleCount THEN
    CopyDetectionCountAndResetDetectionCountInThisCycle();
END_IF

FOR IteratorCounter := 1 TO TotalAsserts BY 1 DO
      IF F_IsAnyEqualToUnionValue(uExpectedOrActual := AssertResultInstances[IteratorCounter].AssertResult.Expected,
                                  ExpectedOrActualSize := ExpectedSize,
                                  ExpectedOrActualTypeClass := ExpectedTypeClass,
                                  ExpectedOrActualValue := ExpectedValue) AND
         F_IsAnyEqualToUnionValue(uExpectedOrActual := AssertResultInstances[IteratorCounter].AssertResult.Actual,
                                  ExpectedOrActualSize := ActualSize,
                                  ExpectedOrActualTypeClass := ActualTypeClass,
                                  ExpectedOrActualValue := ActualValue) AND
        AssertResultInstances[IteratorCounter].AssertResult.Message = Message AND
        AssertResultInstances[IteratorCounter].AssertResult.TestInstancePath = TestInstancePath THEN
        AssertResultInstances[IteratorCounter].DetectionCountThisCycle :=
            AssertResultInstances[IteratorCounter].DetectionCountThisCycle + 1;
            FoundOne := TRUE;
        IF AssertResultInstances[IteratorCounter].DetectionCountThisCycle >
                AssertResultInstances[IteratorCounter].DetectionCount THEN // This assert is new
                AdditionalIdenticalAssert := TRUE;
        END_IF
        EXIT;
    END_IF
END_FOR

(* If not found anything, create the first *)
IF NOT FoundOne THEN
    (* No existing match found, create a new entry *)
    AddAssertResult(ExpectedSize := ExpectedSize,
                    ExpectedTypeClass := ExpectedTypeClass,
                    ExpectedValue := ExpectedValue,
                    ActualSize := ActualSize,
                    ActualTypeClass := ActualTypeClass,
                    ActualValue := ActualValue,
                    Message := Message, TestInstancePath := TestInstancePath);

    CreateAssertResultInstance(ExpectedSize := ExpectedSize,
                               ExpectedTypeClass := ExpectedTypeClass,
                               ExpectedValue := ExpectedValue,
                               ActualSize := ActualSize,
                               ActualTypeClass := ActualTypeClass,
                               ActualValue := ActualValue,
                               Message := Message, TestInstancePath := TestInstancePath);
(* An additional instance of this assert needs to be created *)
ELSIF AdditionalIdenticalAssert THEN
    AddAssertResult(ExpectedSize := ExpectedSize,
                    ExpectedTypeClass := ExpectedTypeClass,
                    ExpectedValue := ExpectedValue,
                    ActualSize := ActualSize,
                    ActualTypeClass := ActualTypeClass,
                    ActualValue := ActualValue,
                    Message := Message, TestInstancePath := TestInstancePath);
(* In all other cases, this assert has already been reported, we don't need to do anything *)
ELSE
    AlreadyReported := TRUE;
END_IF

(* Update the cycle count *)
CycleCount := TwinCAT_SystemInfoVarList._TaskInfo[GetCurrentTaskIndex.index].CycleCount;
END_METHOD

END_FUNCTION_BLOCK

// POUs/FB_FileControl
(*
    This functionblock can open, close, read, write and delete files on the local filesystem
*)
FUNCTION_BLOCK FB_FileControl
VAR
    FileAccessMode : SysFile.ACCESS_MODE := SysFile.AM_APPEND_PLUS; // Append_Plus creates the file if it doesn't exist yet. 
    FileHandle : SysFile.SysTypes.RTS_IEC_HANDLE;
END_VAR

(*
    Closes the current opened file.
*)
METHOD PUBLIC Close : SysFile.SysTypes.RTS_IEC_RESULT;
IF FileHandle <> SysFile.SysTypes.RTS_INVALID_HANDLE THEN
    Close := SysFile.SysFileClose(hFile := FileHandle);
ELSE
    Close := SysDir.CmpErrors.Errors.ERR_INVALID_HANDLE;
END_IF
END_METHOD

(*
    Deletes a file specified by name, if it exists.
*)
METHOD PUBLIC Delete : SysFile.SysTypes.RTS_IEC_RESULT;
VAR_INPUT
    (* File name can contain an absolute or relative path to the file. Path entries must be separated with a forward slash (/) *)
    FileName : Tc2_System.T_MaxString;
END_VAR
Delete := SysFile.SysFileDelete(szFileName := FileName);
END_METHOD

(*
    Opens a file
*)
METHOD PUBLIC Open : SysFile.SysTypes.RTS_IEC_RESULT;
VAR_INPUT
    FileName : Tc2_System.T_MaxString := 'filepath/output.xml';  // File name can contain an absolute or relative path to the file. Path entries must be separated with a Slash (/)
    FileAccessMode : SysFile.ACCESS_MODE := SysFile.ACCESS_MODE.AM_APPEND_PLUS;
END_VAR
FileHandle := SysFile.SysFileOpen(szFile := Filename,
                                  am := FileAccessMode,
                                  pResult := ADR(Open));
END_METHOD

(*
    Reads a file from disk into the buffer
*)
METHOD Read : SysFile.SysTypes.RTS_IEC_RESULT;
VAR_INPUT
    BufferPointer : POINTER TO BYTE; // Call with ADR();
    Size : UDINT; // Call with SIZEOF(); 
END_VAR
VAR_OUTPUT
    FileSize : SysFile.SysTypes.RTS_IEC_SIZE;
END_VAR
IF FileHandle <> SysFile.SysTypes.RTS_INVALID_HANDLE THEN
    FileSize := SysFile.SysFileRead(hFile := FileHandle, 
                                    pbyBuffer := BufferPointer,
                                    ulSize := Size,
                                    pResult := ADR(Read));
ELSE
    Read := SysDir.CmpErrors.Errors.ERR_INVALID_HANDLE;                  
END_IF
END_METHOD

(* 
    Writes the contents of the buffer into a file.
*)
METHOD Write : SysFile.SysTypes.RTS_IEC_RESULT;
VAR_INPUT
    BufferPointer : POINTER TO BYTE; // Call with ADR();
    Size : UDINT; // Call with SIZEOF();
END_VAR
IF FileHandle <> SysFile.SysTypes.RTS_INVALID_HANDLE THEN
    SysFile.SysFileWrite(hFile := FileHandle,
                         pbyBuffer := BufferPointer,
                         ulSize := Size,
                         pResult := ADR(Write));
ELSE
    Write := SysDir.CmpErrors.Errors.ERR_INVALID_HANDLE;                  
END_IF
END_METHOD

END_FUNCTION_BLOCK

// POUs/FB_StreamBuffer
(*
    This functionblock acts as a stream buffer for use with FB_XmlControl
*)
FUNCTION_BLOCK FB_StreamBuffer 
VAR
    _PointerToStringBuffer : POINTER TO BYTE;
    _BufferSize : UDINT;
    _Length : UDINT;
END_VAR

(*
    Appends a string to the buffer
*)
PROPERTY Append : Tc2_System.T_MaxString
SET
VAR
    ByteIn : POINTER TO BYTE;
    ByteBuffer : POINTER TO BYTE;
END_VAR
ByteIn := ADR(Append); 
ByteBuffer := _PointerToStringBuffer + _Length; // set start address

WHILE ByteIn^ <> 0 AND (_Length < _BufferSize ) DO
    ByteBuffer^ := ByteIn^; //Copy the 1st byte
    _Length := _Length + 1; // set new buffer length
    ByteIn := ByteIn + 1; // calculate new start address 
    ByteBuffer := ByteBuffer + 1; // calculate new start address 
END_WHILE;

ByteBuffer := _PointerToStringBuffer + _Length; // String End
ByteBuffer^ := 0; // null terminated string
END_SET
END_PROPERTY

(*
    Read current Buffersize
*)
PROPERTY BufferSize : UDINT
GET
BufferSize := _BufferSize;
END_GET
END_PROPERTY

(*  
    Clears the buffer and sets the length to 0
*)
METHOD PUBLIC Clear
VAR
	Count : UDINT;
END_VAR
IF (_PointerToStringBuffer = 0) OR (_BufferSize = 0) THEN
    RETURN;
END_IF

FOR Count := 0 TO (_BufferSize - 1) DO
    _PointerToStringBuffer[Count] := 0;
END_FOR

_Length := 0;
END_METHOD

(*
    Copies a string from the character buffer
*)
METHOD PUBLIC Copy : Tc2_System.T_MaxString
VAR_INPUT
    StartPos : UDINT;
    EndPos : UDINT;
END_VAR
VAR_OUTPUT
    CopyLen : UDINT;
    XmlError : E_XmlError;
END_VAR
VAR
    Loop : UDINT;
    PointerToByteToCopy : POINTER TO BYTE;
    PointerToBuffer : POINTER TO BYTE;
    CurPos : UDINT;
END_VAR
Loop := 0;
PointerToByteToCopy := ADR(Copy);
PointerToBuffer := _PointerToStringBuffer + StartPos - 1;

WHILE(Loop < SIZEOF(Copy)) AND (StartPos - 1 + Loop < _Length) AND (StartPos + Loop < EndPos) DO
    PointerToByteToCopy^ := PointerToBuffer^;
    Loop := Loop + 1;
    PointerToByteToCopy := ADR(Copy) + Loop;
    PointerToBuffer := _PointerToStringBuffer + StartPos + Loop -1;
END_WHILE;

IF Loop = SIZEOF(Copy) THEN
    XmlError := E_XmlError.ErrorStringLen;
ELSIF StartPos - 1 + Loop = _Length THEN
    XmlError := E_XmlError.ErrorMaxBufferLen;
ELSE
    XmlError := E_XmlError.OK;
END_IF;

PointerToByteToCopy^ := 0;
CopyLen :=  Loop;
END_METHOD

METHOD PUBLIC CutOff : Tc2_System.T_MaxString
VAR_INPUT
    StartPos : UDINT;
END_VAR
VAR_OUTPUT
    CutLen : UDINT; 
    XmlError : E_XmlError;
END_VAR
VAR
    Loop : UDINT;
    PointerToByteToCut : POINTER TO BYTE;
    PointerToByteBuffer : POINTER TO BYTE;
END_VAR
Loop := 0;
PointerToByteToCut := ADR(CutOff);
PointerToByteBuffer := _PointerToStringBuffer + StartPos - 1;

WHILE PointerToByteBuffer^ <> 0 AND(Loop < SIZEOF(CutOff)) AND StartPos -1  + Loop < _Length DO
    PointerToByteToCut^ := PointerToByteBuffer^;
    Loop := Loop + 1;
    PointerToByteToCut := ADR(CutOff) + Loop;
    PointerToByteBuffer := _PointerToStringBuffer + StartPos - 1 + Loop;
END_WHILE;

IF PointerToByteBuffer^ = 0 THEN
    XmlError := E_XmlError.OK;
ELSIF Loop = SIZEOF(CutOff) THEN
    XmlError := E_XmlError.ErrorStringLen;
ELSIF StartPos - 1 + Loop = _Length THEN
    XmlError := E_XmlError.ErrorMaxBufferLen;
END_IF;

PointerToByteToCut^ := 0;
_Length := StartPos -1;

PointerToByteBuffer := _PointerToStringBuffer + StartPos - 1;
PointerToByteBuffer^ := 0;

CutLen := Loop;
END_METHOD

(* 
    Find a searchstring in the buffer and returns its position.
    It's possible to add a preffered startposition within buffer
*)
METHOD PUBLIC Find : UDINT
VAR_INPUT
    SearchString : STRING;
    StartPos : UDINT;
END_VAR
VAR
    Loop : UDINT;
    Search : UDINT;
    PointerToBuffer : POINTER TO BYTE;
    PointerToSearch : POINTER TO BYTE;
END_VAR
Loop := 0;
Search := 0;

PointerToBuffer := _PointerToStringBuffer + StartPos;
PointerToSearch := ADR(SearchString);

